(* CODESYS project cyber-gprs.20190329.3.project

Project tree, tasks and I/O mapping:
  Changsha_Xiangji_ARM_Cortex_A9_xilinx_zynq7000_linux : Changsha Xiangji-ARM Cortex A9(xilinx zynq7000)-linux, Changsha Xiangji Hiden Technology Co.Ltd, version 3.5.10.40
    application Application
      libraries: CAA Types Extern, 3.5.10.0 (CAA Technical Workgroup); VisuDialogs, * (System); CAA Real Time Clock Extern, 3.5.10.0 (CAA Technical Workgroup); CAA Callback Extern, 3.5.11.0 (CAA Technical Workgroup); CAA Can Low Level Extern, 3.5.11.0 (CAA Technical Workgroup); CAA Can Low Level Imp Extern, 3.5.11.0 (CAA Technical Workgroup); SysMem, 3.5.12.0 (System); CAA Net Base Services, 3.5.12.0 (CAA Technical Workgroup); CAA SerialCom, 3.5.12.0 (CAA Technical Workgroup); CAA File, 3.5.12.0 (CAA Technical Workgroup); CAA DTUtil Extern, 3.5.12.0 (CAA Technical Workgroup); SysFile, 3.5.9.0 (System); SysTypes2 Interfaces, * (System); Standard, * (System); cyber gpio, 3.5.10.40 (cyber); Util, * (System)
      task Task (cyclic, interval 50 ms, priority 0) calls prg_main
      task task_can (cyclic, interval 50 ms, priority 5) calls prg_can0, prg_can1, prg_test_can
      task EtherCAT_Task (cyclic, interval 10 ms, priority 1) calls nothing
      task VISU_TASK (cyclic, interval 100 ms, priority 31) calls VisuElems.Visu_Prg
      task Task_gprs (cyclic, interval 20 ms, priority 1) calls prg_heartbeat
      CAN_COMM/
        program prg_can0 [ST]: set_buf_18004f07, set_buf_18074f07, get_buf_0c00074f, proc_screen_data, set_buf_18104f07, set_buf_0801EE2A, get_buf_0C112AEE, set_buf_18114f07, set_buf_18044f07, set_buf_18024f07, set_buf_18014f07, get_buf_0c02074f, get_buf_0C132AEE, get_buf_0c05074f, get_buf_0c04074f, set_buf_18054f07, get_buf_0c01074f, get_buf_0C122AEE, set_buf_18124f07, set_buf_18084f07, set_buf_18064f07, set_buf_18144f07, set_buf_18094f07, set_buf_18034f07, set_buf_18134f07, get_buf_0c03074f, get_buf_0c07074f, get_buf_0c06074f
        program prg_can1 [ST]
        program prg_test_can [ST]
        function CAN_Send_MSG [ST]
      visualisation main
      program Test [ST]
      program Falsh_RW [ST]
      parameters/
        function fn_write_para_file [ST]
        function fn_read_para_file [ST]
        data type ST_PARA
      program prg_main [ST]
      global variables GVL
      funcs/
        function block FB_DOH_FAULT [ST]
        function is_hex [ST]
      program DO_fault [ST]
      GPRS/
        function block File_Read [ST]
        function Iccid_Get [ST]
        function block Packet_Heart [ST]
        program prg_heartbeat [ST]
        function block fb_get_iccid [ST]
        function block fb_m26 [ST]
        function block fb_get_lac [ST]
        function fn_cyber_layer1 [ST]
        function fn_cyber_layer2 [ST]
        function fn_cyber_heartBeat [ST]
        function fn_sn_str_to_byte [ST]
      gprs_lib/
        function block Com_Read [ST]
        function block reset_gprs [ST]
        function block Udp_Config [ST]
        function block Udp_Init [ST]
        function block UDP_Read [ST]
        function block Udp_Write [ST]
    IoDrvMIC7001 : IoDrvMIC7001, Cyber-MI, version 18.11.1
        input  Application.ai_20 : DWORD  // Ai20-Do02@C13
        input  Application.ai_21 : DWORD  // Ai21-Do03@C01
        input  Application.ai_22 : DWORD  // Ai22-Do04@C03
        input  Application.ai_23 : DWORD  // Ai23-Do05@C04
        input  Application.ai_24 : DWORD  // Ai24-Do06@C05
        input  Application.ai_25 : DWORD  // Ai25-Do07@C06
        input  Application.ai_26 : DWORD  // Ai26-Do08@C08
        input  Application.ai_27 : DWORD  // Ai27-Do09@C09
        input  Application.ai_28 : DWORD  // Ai28-Do10@C10
        input  Application.ai_29 : DWORD  // Ai29-Do11@C11
        input  Application.ai_30 : DWORD  // Ai30-Do12@D34
        input  Application.ai_31 : DWORD  // Ai31-Do13@D35
        input  Application.ai_34 : DWORD  // Ai34-Do16@D10
        input  Application.ai_35 : DWORD  // Ai35-Do17@D09
        input  Application.ai_36 : DWORD  // Ai36-Do18@D08
        input  Application.ai_37 : DWORD  // Ai37-Do19@D07
        input  Application.ai_38 : DWORD  // Ai38-Do20@D05
        input  Application.ai_39 : DWORD  // Ai39-Do21@D04
        input  Application.ai_40 : DWORD  // Ai40-Do22@D03
        input  Application.ai_41 : DWORD  // Ai41-Do23@D02
        input  Application.DI_cleanwater_LOW : DWORD  // Ai46-Ao00@C22
        input  Application.DI_Totvalve_Open : BOOL  // Di00-Ai00@C16
        input  Application.DI_water_overflow : BOOL  // Di02-Ai02@C17
        input  Application.DI_fog_pump_press_ok : BOOL  // Di05-Ai05@C19
        input  Application.DI_air_press_low : BOOL  // Di06-Ai06@C31
        input  Application.DI_Hpre_valve_open : BOOL  // Di07-Ai07@C20
        input  Application.DI_box_door_close : BOOL  // Di08-Ai08@C18
        input  Application.DI_backup_power_open : BOOL  // Di09-Ai09@D18
        input  Application.DI_Sweep_Down : BOOL  // Di10-Ai10@D20
        input  Application.DI_Rod_noDown : BOOL  // Di11-Ai11@D31
        input  Application.DI_Sweep_Up : BOOL  // Di12-Ai12@D19
        input  Application.DI_auxiliary2_warte_H : BOOL  // Di13-Ai13@D30
        input  Application.DI_auxiliary1_warte_H : BOOL  // Di14-Ai14@D29
        input  Application.DI_oil_release_valve : BOOL  // Di16-Ai16@D28
        input  Application.DI_Rcar : BOOL  // Di17-Ai17@D16
        input  Application.DI_oil_filter_block : BOOL  // Di18-Ai18@C25
        input  Application.DI_oil_level_low : BOOL  // Di19-Ai19@C24
        input  Application.DI_power_on : BOOL  // Di32-Ai32@D23
        input  Application.DI_sweep_out : BOOL  // Di33-Ai33@D12
        input  Application.DI_wastewater_full : BOOL  // Di42-Ai42@C23
        input  Application.DI_sweep_return : BOOL  // Di45-Ai45@D13
        output Application.DO_pointshoot_down : BOOL  // Do02-Ai20@C13
        output Application.DO_Lsweep_down : BOOL  // Do03-Ai21@C01
        output Application.DO_Lsweep_up : BOOL  // Do04-Ai22@C03
        output Application.DO_Rsweep_down : BOOL  // Do05-Ai23@C04
        output Application.DO_Rsweep_up : BOOL  // Do06-Ai24@C05
        output Application.DO_Lsweep_out : BOOL  // Do07-Ai25@C06
        output Application.DO_Rsweep_out : BOOL  // Do08-Ai26@C08
        output Application.DO_Lrod_out : BOOL  // Do09-Ai27@C09
        output Application.DO_Rrod_out : BOOL  // Do10-Ai28@C10
        output Application.DO_pointshoot_up : BOOL  // Do11-Ai29@C11
        output Application.DO_backup_power : BOOL  // Do12-Ai30@D34
        output Application.DO_Motor_en : BOOL  // Do13-Ai31@D35
        output Application.DO_fog_Spump : BOOL  // Do16-Ai34@D10
        output Application.DO_Hpre_pump : BOOL  // Do17-Ai35@D09
        output Application.DO_selfclean_water : BOOL  // Do18-Ai36@D08
        output Application.DO_Hpressure_water : BOOL  // Do19-Ai37@D07
        output Application.DO_Suction_water : BOOL  // Do20-Ai38@D05
        output Application.DO_Rrod_water : BOOL  // Do21-Ai39@D04
        output Application.DO_Lrod_water : BOOL  // Do22-Ai40@D03
        output Application.DO_water_overflow : BOOL  // Do23-Ai41@D02
        output Application.DO_pointshoot_left : BOOL  // Do28-Pwmi00@C33
        output Application.DO_pointshoot_right : BOOL  // Do29-Pwmi01@C34
        output Application.DO_watercooler_pump : BOOL  // Do30-Pwmi02@D25
        output Application.DO_cooler_fan : BOOL  // Do31-Pwmi03@D26
        unmapped channels: Ai00@C16, Ai01@C28, Ai02@C17, Ai03@C29, Ai04@C30, Ai05@C19, Ai06@C31, Ai07@C20, Ai08@C18, Ai09@D18, Ai10@D20, Ai11@D31, Ai12@D19, Ai13@D30, Ai14@D29, Ai15@D17, Ai16@D28, Ai17@D16, Ai18-Do00@C25, Ai19-Do01@C24, Ai32-Do14@D23, Ai33-Do15@D12, Ai42-Do24@C23, Ai43-Do25@C35, Ai44-Do26@D24, Ai45-Do27@D13, Ai47-Ao01@D14, Ai48_Pi02, Ai49_Out5V, Ai50_VCC, Ai51_VCC_L, Ai52_VCC_R, Ai53_Pwm-i0, Ai54_Pwm-i1, Ai55_Pwm-i2, Ai56_Pwm-i3, Ai57_CPU-T, Ai58_G-x, Ai59_G-y, Ai60_G-z,
          Ai61-reserved, Ai62-IO-cntr, Ai63-CDS-cntr, Di01-Ai01@C28, Di03-Ai03@C29, Di04-Ai04@C30, Di15-Ai15@D17, Di20-Ai20@C13, Di21-Ai21@C01, Di22-Ai22@C03, Di23-Ai23@C04, Di24-Ai24@C05, Di25-Ai25@C06, Di26-Ai26@C08, Di27-Ai27@C09, Di28-Ai28@C10, Di29-Ai29@C11, Di30-Ai30@D34, Di31-Ai31@D35, Di34-Ai34@D10, Di35-Ai35@D09, Di36-Ai36@D08, Di37-Ai37@D07, Di38-Ai38@D05, Di39-Ai39@D04, Di40-Ai40@D03, Di41-Ai41@D02, Di43-Ai43@C35, Di44-Ai44@D24, Di46-Ai46@C22, Di47-Ai47@D14, Di48-Pi00@C15, Di49-Pi01@C14, Di50-Pi02@D22, Di51-Pi03@D21, Di52-reserved, Di53-reserved, Di54-reserved, Di55-reserved, Di56-reserved,
          Di57-reserved, Di58-reserved, Di59-reserved, Di60-reserved, Di61-reserved, Di62-reserved, Di63-reserved, Pi00-Di48@C15, Pi01-Di49@C14, Pi02-Di50@D22, Pi03-Di51@D21, Do00-Ai18@C25, Do01-Ai19@C24, Do14-Ai32@D23, Do15-Ai33@D12, Do24-Ai42@C23, Do25-Ai43@C35, Do26-Ai44@D24, Do27-Ai45@D13, PWM00@C25, PWM01@C24, PWM02@C13, PWM03@C01, PWM04@C03, PWM05@C04, PWM06@C05, PWM07@C06, PWM08@C08, PWM09@C09, PWM10@C10, PWM11@C11, PWM12@D34, PWM13@D35, PWM14@D23, PWM15@D12, PWM16@D10, PWM17@D09, PWM18@D08, PWM19@D07, PWM20@D05,
          PWM21@D04, PWM22@D03, PWM23@D02, PWM24@C23, PWM25@C35, PWM26@D24, PWM27@D13, PWM28-Pwmi00@C33, PWM29-Pwmi01@C34, PWM30-Pwmi02@D25, PWM31-Pwmi03@D26, PWM_I_0@C33, PWM_I_1@C34, PWM_I_2@D25, PWM_I_3@D26, Ao00-Ai46@C22, Ao01-Ai47@D14, LED_run, LED_err, LED_usr, ctrl_ai_raw, ctrl_adjust, ctrl_adj0, ctrl_adj1, ctrl_adj2, ctrl_adj3, ctrl_adj4
    SoftMotion General Axis Pool
    EtherCAT_Master_SoftMotion : EtherCAT Master SoftMotion, 3S - Smart Software Solutions GmbH, version 3.5.12.40
        settings: MasterCycleTime = 10000; SlaveAutoRestart = True; NetworkName = 'eth0'; NetworkName = "eth0"; SelectNetworkByName = True; SrcAddress1 = 29185; SrcAddress2 = 102470395
      MIR3501 : MIR3501, xiangrui, order no. MIR3501, version Revision=16#00000000
          settings: StationAlias = 0; DC sync0 cycletime = 10000; DC sync1 cycletime = 10000
          output Application.DO_wastewater_valve : BIT  // DO-00-C01
          output Application.DO_wastewater_pump : BIT  // DO-01-C02
          output Application.DO_oil_release_valve : BIT  // DO-02-C03
          output Application.DO_Sweep_Mspeed : BIT  // DO-03-C04
          output Application.DO_Sweep_Lspeed : BIT  // DO-04-C05
          output Application.DO_RSweep : BIT  // DO-05-C06
          output Application.DO_LASweep : BIT  // DO-06-C07
          output Application.DO_RASweep : BIT  // DO-07-C08
          output Application.DO_Box_Down : BIT  // DO-08-C09
          output Application.DO_Suction_Down : BIT  // DO-10-C11
          output Application.DO_Suction_Up : BIT  // DO-11-C12
          output Application.DO_Door_Close : BIT  // DO-12-C26
          output Application.DO_Door_Open : BIT  // DO-13-C25
          output Application.DO_Box_Up : BIT  // DO-15-C33
          unmapped channels: DO-09-C10, DO-14-C34, PWM-00-C26, PWM-01-C25, PWM-02-C34, PWM-03-C33, PWMi-00-C26, PWMi-01-C25, PWMi-02-C34, PWMi-03-C33, AI-00-C17, AI-01-C29, AI-02-C18, AI-03-C30, AI-04-C14, AI-05-C15, AI-06-C21, AI-07-C22, AI-08-C01, AI-09-C02, AI-10-C03, AI-11-C04, AI-12-C05, AI-13-C06, AI-14-C07, AI-15-C08, AI-16-C09, AI-17-C10, AI-18-C11, AI-19-C12, AI-20, AI-21, AI-22, AI-23, DI-00-C17, DI-01-C29, DI-02-C18, DI-03-C30, DI-04-C14, DI-05-C15,
            DI-06-C21, DI-07-C22, DI-08-C01, DI-09-C02, DI-10-C03, DI-11-C04, DI-12-C05, DI-13-C06, DI-14-C07, DI-15-C08, DI-16-C09, DI-17-C10, DI-18-C11, DI-19-C12, DI-20-C27, DI-21-C16, DI-22-C19, DI-23-C20, DI-24, DI-25, DI-26, DI-27, DI-28, DI-29, DI-30, DI-31, PI-00-C27, PI-01-C16, PI-02-C19, PI-03-C20
  5ce3da45-db07-42e7-a21c-a00fff4ed8f6|C:\Users\Administrator\Desktop\robotview1.bmp
  5ce3da45-db07-42e7-a21c-a00fff4ed8f6|C:\Users\Administrator\Desktop\robotview2.bmp
  text list GlobalTextList
  5ce3da45-db07-42e7-a21c-a00fff4ed8f6|C:\Users\Administrator\Desktop\1129.bmp
  5ce3da45-db07-42e7-a21c-a00fff4ed8f6|C:\Users\Administrator\Desktop\robotview0.bmp
*)

// Changsha_Xiangji_ARM_Cortex_A9_xilinx_zynq7000_linux/Application/parameters/ST_PARA
TYPE ST_PARA :
STRUCT
	len:UINT := 64;   //参数的个数，根据需要设置。设置后最好不变，改变后以前保存的参数作废
	para_val:ARRAY[0..63] OF REAL; 	
	para_ok:BOOL := FALSE;
END_STRUCT
END_TYPE

// Changsha_Xiangji_ARM_Cortex_A9_xilinx_zynq7000_linux/Application/GVL
VAR_GLOBAL
	g_parameters: ST_PARA;	
	
	//通过CAN总线从底盘读到的信息
	High_voltage_Ready:BOOL := FALSE;
	Chassis_speed:BYTE := 0;
	Chassis_Soc:BYTE := 0;
//********以下为显示屏下发指令*********//
    // 全洗扫
	HMI_Awashsweep: BOOL := FALSE;	
    // 左洗扫
	HMI_Lwashsweep: BOOL := FALSE;	
    // 右洗扫
	HMI_Rwashsweep: BOOL := FALSE;
	// 全扫路
	HMI_Asweeproad: BOOL := FALSE;
	// 左扫路
	HMI_Lsweeproad: BOOL := FALSE;
	// 右扫路
	HMI_Rsweeproad: BOOL := FALSE;
	// 全清洗
	HMI_Acleanwash: BOOL := FALSE;
	// 右清洗
	HMI_Lcleanwash: BOOL := FALSE;
	// 右全洗
	HMI_Rcleanwash: BOOL := FALSE;
	// 停扫
	HMI_stop_sweep: BOOL := FALSE;
	// 电机启动
	HMI_start_motor: BOOL := FALSE;
	// 电机停止
	HMI_stop_motor: BOOL := FALSE;
	// 速度加
	HMI_Inc_Speed: BOOL := FALSE;
	// 速度减
	HMI_Dec_Speed: BOOL := FALSE;
	// 标准转速
	HMI_Standard_speed: BOOL := FALSE;
	// 强力转速
	HMI_Strong_speed: BOOL := FALSE;
	// 箱门关
	HMI_Door_Close: BOOL := FALSE;
	// 箱门开
	HMI_Door_Open: BOOL := FALSE;
	// 箱体升
	HMI_Box_Up: BOOL := FALSE;
	// 箱体降
	HMI_Box_Down: BOOL := FALSE;
	// 喷雾降尘泵
	HMI_fog_Spump: BOOL := FALSE;
	// 自洁
	HMI_selfclean: BOOL := FALSE;
	// 污水泵
	HMI_wastewater_pump: BOOL := FALSE;
	// 扫盘高速
	HMI_Sweep_Hspd: BOOL := FALSE;
	// 扫盘中速
	HMI_Sweep_Mspd: BOOL := FALSE;
	// 扫盘低速
	HMI_Sweep_Lspd: BOOL := FALSE;
	// 高压冲洗
	HMI_Hpre_wash: BOOL := FALSE;
	// 点喷上
	HMI_pointshoot_up: BOOL := FALSE;
	// 点喷下
	HMI_pointshoot_down: BOOL := FALSE;
	// 点喷左
	HMI_pointshoot_left: BOOL := FALSE;
	// 点喷右
	HMI_pointshoot_right: BOOL := FALSE;
	// 排水启动
	HMI_drain_start: BOOL := FALSE;
	// 排水自动
	HMI_drain_auto: BOOL := FALSE;
	// 排水手动
	HMI_drain_manual: BOOL := FALSE;
	// 左喷杆排水
	HMI_Lrod_drain: BOOL := FALSE;
	// 右喷杆排水
	HMI_Rrod_drain: BOOL := FALSE;
	// 高辅排水
	HMI_Hpressure_drain: BOOL := FALSE;
	// 自洁排水
	HMI_selfclean_drain: BOOL := FALSE;
	// 吸嘴排水
	HMI_Suction_drain: BOOL := FALSE;
	// 功能测试
	HMI_func_test: BOOL := FALSE;
	// 更换扫刷
	HMI_replace_Sweep: BOOL := FALSE;
	// 智能
	HMI_intelligent: BOOL := FALSE;
	// 清洁
	HMI_cleanly: BOOL := FALSE;
	// 一般
	HMI_normal: BOOL := FALSE;
	// 污染
	HMI_dirty: BOOL := FALSE;
	// 水冷泵测试
	Test_watercooler_pump: BOOL := FALSE;
	// 散热风扇测试
	Test_cooler_fan: BOOL := FALSE;
	// 扫盘中速
	Test_Sweep_Mspeed: BOOL := FALSE;
	// 扫盘低速
	Test_Sweep_Lspeed: BOOL := FALSE;
	// 左扫旋转
	Test_LSweep: BOOL := FALSE;
	// 右扫旋转
	Test_RSweep: BOOL := FALSE;
	// 全扫旋转
	Test_ASweep: BOOL := FALSE;
	// 箱体降
	Test_Box_Down: BOOL := FALSE;
	// 箱体升
	Test_Box_Up: BOOL := FALSE;
	// 吸嘴下降
	Test_Suction_Down: BOOL := FALSE;
	// 吸嘴上升
	Test_Suction_Up: BOOL := FALSE;
	// 箱门开
	Test_Door_Open: BOOL := FALSE;
	// 箱门关
	Test_Door_Close: BOOL := FALSE;
	// 左扫盘下降
	Test_LSweep_Down: BOOL := FALSE;
	// 左扫盘上升
	Test_LSweep_Up: BOOL := FALSE;
	// 右扫盘下降
	Test_RSweep_Down: BOOL := FALSE;
	// 右扫盘上升
	Test_RSweep_Up: BOOL := FALSE;
	// 左扫盘摆出
	Test_LSweep_out: BOOL := FALSE;
	// 右扫盘摆出
	Test_RSweep_out: BOOL := FALSE;
	// 左喷杆摆出
	Test_Lrod_OUT: BOOL := FALSE;
	// 右喷杆摆出
	Test_Rrod_OUT: BOOL := FALSE;
	// 左喷杆喷水
	Test_Lrod_water: BOOL := FALSE;
	// 右喷杆喷水
	Test_Rrod_water: BOOL := FALSE;
	// 吸嘴喷杆喷水
	Test_Suction_water: BOOL := FALSE;
	// 高压喷杆喷水
	Test_Hpre_wash: BOOL := FALSE;
	// 自洁
	Test_selfclean: BOOL := FALSE;
	// 高压水泵啮合
	Test_Hpre_pump_gearin: BOOL := FALSE;
	// 喷雾降尘泵
	Test_fogpump: BOOL := FALSE;
	// 点喷上
	Test_pointshoot_up: BOOL := FALSE;
	// 点喷下
	Test_pointshoot_down: BOOL := FALSE;
	// 点喷左
	Test_pointshoot_left: BOOL := FALSE;
	// 点喷右
	Test_pointshoot_right: BOOL := FALSE;
	// 污水泵
	Test_wastewater_pump: BOOL := FALSE;
	// 污水球阀
	Test_wastewater_valve: BOOL := FALSE;
	// 备用动力打开
	Test_backup_power: BOOL := FALSE;
	// 转速加减值
	Re_IncDec_Speed: UINT;
	// 电机最低转速
	Re_motor_min_speed: UINT;
	// 标准转速
	Re_normal_speed: UINT;
	// 强力转速
	Re_strong_Speed: UINT;
	// 扫盘转速
	Re_Sweep_Speed: UINT;
	// 高压水泵超速报警
	Re_Pumpspeed_arm: UINT;
	// 高压水泵超速停止
	Re_Pumpspeed_stop: UINT;
	// 电机最高转速
	Re_MAX_Speed: UINT;
	// 电机怠速
	Re_Idle_Speed: UINT;	
    // 清洁低速
	Re_clean_low_speed: UINT;
	// 清洁中低速
	Re_clean_midlow_speed: UINT;
	// 清洁中高速
	Re_clean_midhigh_speed: UINT;
	// 清洁高速
	Re_clean_high_speed: UINT;
	// 一般低速
	Re_normal_low_speed: UINT;
	// 一般中低速
	Re_normal_midlow_speed: UINT;
	// 一般中高速
	Re_normal_midhigh_speed: UINT;
	// 一般高速
	Re_normal_high_speed: UINT;
	// 污染低速
	Re_dirty_low_speed: UINT;
	// 污染中低速
	Re_dirty_midlow_speed: UINT;
	// 污染中高速
	Re_dirty_midhigh_speed: UINT;
	// 污染高速
	Re_dirty_high_speed: UINT;
	//************************************
	//********以下为控制器输出**********//
	//***********************************
	// 左扫盘下降
	DO_Lsweep_down: BOOL;
	// 左扫盘上升
	DO_Lsweep_up: BOOL;
	// 右扫盘下降
	DO_Rsweep_down: BOOL;
	// 右扫盘上升
	DO_Rsweep_up: BOOL;
	// 左扫盘摆出
	DO_Lsweep_out: BOOL;
	// 右扫盘摆出
	DO_Rsweep_out: BOOL;
	// 左喷杆摆出
	DO_Lrod_out: BOOL;
	// 右喷杆摆出
	DO_Rrod_out: BOOL;
	// 点喷上
	DO_pointshoot_up: BOOL;
	// 点喷下
	DO_pointshoot_down: BOOL;
	// 点喷左
	DO_pointshoot_left: BOOL;
	// 点喷右
	DO_pointshoot_right: BOOL;
	// 水路卸荷阀
	DO_water_overflow: BOOL;
	// 左喷杆喷水
	DO_Lrod_water: BOOL;
	// 右喷杆喷水
	DO_Rrod_water: BOOL;
	// 吸嘴喷杆喷水
	DO_Suction_water: BOOL;
	// 喷雾喷杆喷水
	DO_Hpressure_water: BOOL;
	// 自洁喷水
	DO_selfclean_water: BOOL;
	// 低压隔膜泵
	DO_fog_Spump: BOOL;
	// 高压水泵啮合
	DO_Hpre_pump: BOOL;
	// 电机使能
	DO_Motor_en: BOOL;
	// 水冷泵打开
	DO_watercooler_pump: BOOL;
	// 散热风扇打开
	DO_cooler_fan: BOOL;
	// 备用动力打开
	DO_backup_power: BOOL;
	// 污水泵球阀打开
	DO_wastewater_valve: BOOL;
	// 污水泵打开
	DO_wastewater_pump: BOOL;
	// 油路卸荷阀
	DO_oil_release_valve: BOOL;
	// 扫盘中速
	DO_Sweep_Mspeed: BOOL;
	// 扫盘低速
	DO_Sweep_Lspeed: BOOL;
	// 右扫旋转
	DO_RSweep: BOOL;
	// 左/全扫旋转
	DO_LASweep: BOOL;
	// 右/全扫旋转
	DO_RASweep: BOOL;
	// 箱体降
	DO_Box_Down: BOOL;
	// 箱体升
	DO_Box_Up: BOOL;
	// 吸盘下降
	DO_Suction_Down: BOOL;
	// 吸盘上升
	DO_Suction_Up: BOOL;
	// 箱门打开
	DO_Door_Open: BOOL;
	// 箱门关闭
	DO_Door_Close: BOOL;
	// 高压水泵啮合
	DO_Hpre_pump1: BOOL;
	// 左扫盘摆出中间变量
	DO_Lsweep_out1: BOOL;
	// 左扫盘下降中间变量
	DO_Lsweep_down1: BOOL;
	// 右扫盘摆出中间变量
	DO_Rsweep_out1: BOOL;
	// 右扫盘下降中间变量
	DO_Rsweep_down1: BOOL;
	// 吸盘下降中间变量
	DO_Suction_Down1: BOOL;
	// 右扫盘上升标志
	DO_Rsweep_up1: BOOL;
	// 吸盘上升标志位
	DO_Suction_Up1: BOOL;
	// 左喷杆摆出标志
	DO_Lrod_out1: BOOL;
	// 右喷杆摆出标志位
	DO_Rrod_out1: BOOL;
	// 喷雾降尘泵标志位
	DO_fog_Spump1: BOOL;
	// 高压冲洗标志位
	DO_Hpressure_water1: BOOL;
	// 自洁标志位
	DO_selfclean_water1: BOOL;
	// 垃圾箱门关标志位
	DO_Door_Close1: BOOL;
	// 垃圾箱门开标志位
	DO_Door_Open1: BOOL;
	// 箱体升标志
	DO_Box_Up1: BOOL;
	// 垃圾箱下降标志
	DO_Box_Down1: BOOL;
	// 水冷泵电机打开标志位
	DO_watercooler_pump_open1: BOOL;
	// 散热风扇打开标志位
	DO_cooler_fan_open1: BOOL;
	
	//********控制器输入**************
	//**********************************
	// 水箱水位低
	DI_cleanwater_LOW: DWORD;
	// 总水阀打开
	DI_Totvalve_Open: BOOL;
	// 箱门关闭
	DI_box_door_close: BOOL;
	// 高压吹净球阀打开
	DI_Hpre_valve_open: BOOL;

	// 污水满
	DI_wastewater_full: BOOL;
	// 撑杆未放下
	DI_Rod_noDown: BOOL;
	// 备用动力开
	DI_backup_power_open: BOOL;
	// 水路卸荷阀卸荷
	DI_water_overflow: BOOL;

	// 电源开关打开
	DI_power_on: BOOL;
	// 倒车
	DI_Rcar: BOOL;
	// 液压卸荷阀
	DI_oil_release_valve: BOOL;
	// 辅污水箱1水位高
	DI_auxiliary1_warte_H: BOOL;
	// 辅污水箱2水位高
	DI_auxiliary2_warte_H: BOOL;
	// 扫盘升
	DI_Sweep_Up: BOOL;
	// 扫盘降
	DI_Sweep_Down: BOOL;
	// 扫盘摆出
	DI_sweep_out: BOOL;
	// 扫盘缩回
	DI_sweep_return: BOOL;
	// 全洗扫标志位
	AwashSweep_HMI: BOOL := FALSE;
	// 左洗扫标志位
	LwashSweep_HMI: BOOL := FALSE;
	// 右洗扫标志位
	RwashSweep_HMI: BOOL := FALSE;
	// 全扫路标志位
	ASweeproad_HMI: BOOL := FALSE;
	// 左扫路标志位
	LSweeproad_HMI: BOOL := FALSE;
	// 右扫路标志位
	RSweeproad_HMI: BOOL := FALSE;
	// 全清洗标志位
	Aclean_HMI: BOOL := FALSE;
	// 左清洗标志位
	Lclean_HMI: BOOL := FALSE;
	// 右清洗标志位
	Rclean_HMI: BOOL := FALSE;
	// 停扫标志位
	Sweep_stop_HMI: BOOL := FALSE;
	// 标准转速标志位
	Standard_speed_HMI: BOOL := FALSE;
	// 强力转速
	Strong_speed_HMI: BOOL := FALSE;
	// 扫盘高速
	Sweep_HSpeed_HMI: BOOL;
	// 扫盘中速
	Sweep_MSpeed_HMI: BOOL;
	// 扫盘低速
	Sweep_LSpeed_HMI: BOOL;
	// 排水启动
	Drain_start_HMI: BOOL := FALSE;
	// 排水自动
	Drain_auto_HMI: BOOL;
	// 排水手动
	Drain_manual_HMI: BOOL;
	// 左喷杆排水
	Lrod_drain_HMI: BOOL;
	// 右喷杆排水
	Rrod_drain_HMI: BOOL;
	// 高辅排水
	Hpressure_drain_HMI: BOOL;
	// 自洁排水
	Selfclean_drain_HMI: BOOL;
	// 吸嘴喷杆排水
	Suction_drain_HMI: BOOL;
	// 更换扫刷标志位
	replace_Sweep_HMI: BOOL;
	// 功能测试
	Func_test_HMI: BOOL;
	// 智能标志位
	Intelligent_HMI: BOOL:= FALSE;
	// 清洁标志位
	Cleanly_HMI: BOOL:= FALSE;
	// 一般标志位
	Normal_HMI: BOOL:= FALSE;
	// 污染标志位
	Dirty_HMI: BOOL:= FALSE;

	// 点喷上标志位
	Pointshoot_up_HMI: BOOL;
	// 点喷下标志位
	Pointshoot_down_HMI: BOOL;
	// 点喷左标志位
	Pointshoot_left_HMI: BOOL;
	// 点喷右标志位
	Pointshoot_right_HMI: BOOL;
	// 水冷泵测试标志位
	cooler_motor_Test: BOOL;
	// 散热风扇测试标志位
	cooler_fan_Test: BOOL;
	// 扫盘中速测试标志位
	Sweep_Mspeed_Test: BOOL;
	// 扫盘低速测试标志位
	Sweep_Lspeed_Test: BOOL;
	// 左扫旋转测试标志位
	LSweep_Test: BOOL;
	// 右扫测试标志位
	RSweep_Test: BOOL;
	// 全扫测试标志位
	ASweep_Test: BOOL;
	// 箱体降测试标志位
	Box_Down_Test: BOOL;
	// 箱体升测试标志位
	Box_Up_Test: BOOL;
	// 吸盘降测试标志位
	Suction_Down_Test: BOOL;
	// 吸盘升测试标志位
	Suction_Up_Test: BOOL;
	// 箱门开测试标志位
	Boxdoor_open_Test: BOOL;
	// 测试标志位
	Boxdoor_close_Test: BOOL;
	// 左扫降测试标志位
	LSweep_Down_Test: BOOL;
	// 左扫升测试标志位
	LSweep_Up_Test: BOOL;
	// 右扫降测试标志位
	RSweep_Down_Test: BOOL;
	// 右扫升测试标志位
	RSweep_Up_Test: BOOL;
	// 左扫摆出测试标志位
	Lrod_OUT_Test: BOOL;
	// 右扫摆出测试标志位
	Rrod_OUT_Test: BOOL;
	// 左喷杆喷水测试标志位
	Lrod_water_Test: BOOL;
	// 右喷杆喷水测试标志位
	Rrod_water_Test: BOOL;
	// 吸嘴喷水测试标志位
	Suction_water_Test: BOOL;
	// 高辅喷水测试标志位
	Hpre_wash_Test: BOOL;
	// 自洁测试标志位
	selfclean_water_Test: BOOL;
	// 高压水泵啮合测试标志位
	Hpress_pump_gearin_Test: BOOL;
	// 喷雾降尘测试标志位
	Fog_pump_Test: BOOL;
	// 左扫摆出测试标志位
	LSweep_out_Test: BOOL;
	// 右扫摆出测试标志位
	RSweep_out_Test: BOOL;
	// 污水泵测试标志位
	Wastewater_pump_Test: BOOL;
	// 污水泵球阀测试标志位
	Wastewater_valve_Test: BOOL;
	// 备用动力测试标志位
	Backup_power_Test: BOOL;
	// 点喷上测试标志位
	Pointshoot_up_Test: BOOL;
	// 点喷下测试标志位
	Pointshoot_down_Test: BOOL;
	// 点喷左测试标志位
	Pointshoot_left_Test: BOOL;
	// 点喷右测试标志位
	Pointshoot_right_Test: BOOL;
	// 电机工作标志位
	Motor_Work: BOOL:= FALSE;
	// 系统工作标志位
	SYS_work: BOOL;
	// 转速加减值
	S_IncDec_Speed: UINT;
	// 电机最低转速
	S_min_speed: UINT;
	// 标准转速
	S_Standard_Speed: UINT;
	// 强力转速
	S_Strong_Speed: UINT;
	// 扫盘转速
	S_Sweep_Speed: UINT;
	// 高压水泵超速报警
	S_Pumpspeed_arm: UINT;
	// 高压水泵超速停止
	S_Pumpspeed_stop: UINT;
	// 最高转速
	S_MAX_Speed: UINT;
	// 电机怠速
	S_Idle_Speed: UINT;
	// 电机实际转矩
	Motor_real_torque_HMI: UINT;
	// 电机实际转速
	Motor_real_speed_HMI: UINT;
	// 电机母线电压
	Motor_bus_voltage_HMI: UINT;
	// 电机相电流
	Motor_phase_current_HMI: UINT;
	// 电机最大允许驱动转矩
	Motor_max_dirve_torque_HMI: UINT;
	// 电机最大允许制动转矩
	Motor_max_brake_torque_HMI: UINT;
	// 电机驱动器温度
	Motor_temp_controller_HMI: BYTE;
	// 电机温度
	Motor_temp_HMI: BYTE;
	// 电机最大转速
	Motor_max_speed_HMI: UINT;
	// 电机运行方向
	Motor_direction_cw: BYTE;
	// 电机工作模式
	Motor_mode: BYTE;
	// 电机状态
	Motor_stat: BYTE;
	// 电机母线欠压
	Motor_bus_low_voltage: BYTE;
	// 电机母线欠压
	Motor_bus_high_voltage: BYTE;
	// 电机控制器过温
	MOtor_ctrller_high_temp: BYTE;
	// 电机过温
	Motor_high_temp: BYTE;
	// 电机IGBT故障
	Motor_igbt_fault: BYTE;
	// 电机超速
	Motor_overspeed: BYTE;
	// 电机通讯故障
	Motor_comm_error: BYTE;
	// 电机过流或短路
	Motor_short: BYTE;
	// 电机堵转故障
	Motor_overload: BYTE;
	// 电机自检故障
	Motor_selfcheck_fault: BYTE;
	// 电机低压供电故障
	Motor_low_voltage: BYTE;
	// 电机传感器故障
	Motor_sensor_fault: BYTE;

	// 设定转速值
	SETspeed_PID: UINT:= 0;
	// 底盘车速
//	Chassis_speed: UINT;
	// 清洁路面低速
	S_clean_low_speed: UINT;
	// 清洁中低速
	S_clean_midlow_speed: UINT;
	// 清洁中高速
	S_clean_midhigh_speed: UINT;
	// 清洁高速
	S_clean_high_speed: UINT;
	// 一般路面低速
	S_normal_low_speed: UINT;
	// 一般路面中低速
	S_normal_midlow_speed: UINT;
	// 一般路面中高速
	S_normal_midhigh_speed: UINT;
	// 一般路面高速
	S_normal_high_speed: UINT;
	// 污染路面低速
	S_dirty_low_speed: UINT;
	// 污染路面中低速
	S_dirty_midlow_speed: UINT;
	// 污染路面中高速
	S_dirty_midhigh_speed: UINT;
	// 污染路面高速
	S_dirty_high_speed: UINT;
	// 水箱水位低报警
	DI_cleanwater_LOW_ALM: BOOL;
	// 请先打开备用动力开关
	Backup_power_Test_warn: BOOL;
	// 水路卸荷阀未关闭故障
	T_water_overflow_noClose: Ton;
	// 水路卸荷阀未打开故障
	T_water_overflow_noOpen: Ton;
	// 喷雾降尘泵压力不正常标志
	T_fog_pump_press_noOk: Ton;
	// 主污水箱水满标志
	T_DI_wastewater_full: Ton;
	// 辅污水箱1水满标志
	T_DI_auxiliary1_warte_H: Ton;
	// 辅污水箱2水满标志
	T_DI_auxiliary2_warte_H: Ton;
	// 污水满故障标志
	Wastewater_full_Fault: BOOL;
	// 辅助水箱水位不一致标志
	T_auxiliary_warte_dif: Ton;
	// 回油过滤堵塞故障标志
	T_DI_oil_filter_block: Ton;
	// 液压油位低故障标志
	T_DI_oil_level_low: Ton;
	// 系统气压低标志
	T_DI_air_press_low: Ton;
	// 倒车标志
	T_DI_Rcar: Ton;
	// 水箱缺水故障标志
	T_DI_cleanwater_LOW: Ton;
	// 高压水泵超速报警
	T_Pumpspeed_H: Ton;
	// 高压水泵超速停止
	T_Pumpspeed_HH: Ton;
	// 请关闭测试提示
	TEST_ALM: BOOL;
	// 倒车提示
	RCAR_ALM: BOOL;
	// 请先打开发动机
	Motor_Work_ALM: BOOL;
	// 倒车故障停机
	DI_Rcar_fault: BOOL;
	// 污水满故障停机
	Wastewater_full_Fault1: BOOL;
	// 底盘电量低于20%
	Chassis_SOC_LOW: BOOL;
	// 底盘电量低7S后停机
	T_Chassis_SOC_LOW: Ton;
	// 隔膜泵球阀未打开
	fog_Spump_arm: BOOL;
	// 污水泵打开标志位
	DO_wastewater_pump_open1: BOOL;
	// 高压水泵未啮合提示
	DO_Hpre_pump_noWork: BOOL;
	// 高压水路球阀未打开提示
	DI_Totvalve_noOpen: BOOL;
	// 高压吹净球阀未打开提示
	DI_Hpre_valve_noOpen: BOOL;
	// 请先打开箱门
	DO_Box_Up_arm: BOOL;
	// 请先放下撑杆
	DO_Box_Down_arm: BOOL;
	// 底盘未上高压提示
	High_voltage_noReady: BOOL;
	// 故障停机
	Fault_STOP: BOOL;
	// 底盘CAN通信故障
	T_Chassis_CAN_fault: TON;
	// 与电机CAN通讯失败
	T_Motor_CAN_fault: Ton;
	// 与屏CAN通讯失败
	T_Screen_CAN_fault: Ton;
	// 屏通讯失败停扫
	HMI_MOTOR_runstop_M: BOOL;
	// 全扫旋转标志
	ASweep: BOOL;
	// 左扫旋转标志
	LSweep: BOOL;
	// 右扫旋转标志
	RSweep: BOOL;
	

	// 喷雾降尘泵压力正常
	DI_fog_pump_press_ok: BOOL;
	// 液压油位低
	DI_oil_level_low: BOOL;
	// 回油过滤堵塞
	DI_oil_filter_block: BOOL;
	// 气路系统压力低
	DI_air_press_low: BOOL;
	Drain_manual_HMI100: BOOL;
	ai_21: DWORD;
	ai_22: DWORD;
	ai_23: DWORD;
	ai_24: DWORD;
	ai_25: DWORD;
	ai_26: DWORD;
	ai_27: DWORD;
	ai_28: DWORD;
	ai_29: DWORD;
	ai_20: DWORD;
	ai_41: DWORD;
	ai_40: DWORD;
	ai_39: DWORD;
	ai_38: DWORD;
	ai_37: DWORD;
	ai_36: DWORD;
	ai_35: DWORD;
	ai_34: DWORD;
	ai_31: DWORD;
	ai_30: DWORD;
					
	DO_Lsweep_down_short: BOOL:= FALSE;  //左扫盘降短路标志
	DO_Lsweep_down_open: BOOL := FALSE;   //左扫盘降开路标志
	DO_Lsweep_up_short: BOOL := FALSE;  // 左扫盘升短路标志
	DO_Lsweep_up_open: BOOL := FALSE;   //左扫盘升开路标志
	DO_Rsweep_down_short: BOOL:= FALSE; //右扫盘降短路
	DO_Rsweep_down_open: BOOL:= FALSE; //右扫盘降开路
	DO_Rsweep_up_short: BOOL:= FALSE; //右扫盘升短路
	DO_Rsweep_up_open: BOOL:= FALSE; //右扫盘升开路
	DO_Lsweep_out_short: BOOL:= FALSE; //左扫摆出短路
	DO_Lsweep_out_open: BOOL:= FALSE; //左扫摆出开路
	DO_Rsweep_out_short: BOOL:= FALSE; //右扫盘摆出短路
	DO_Rsweep_out_open: BOOL:= FALSE; //右扫盘摆出开路
	DO_Lrod_out_short: BOOL:= FALSE; //左喷杆摆出短路
	DO_Lrod_out_open: BOOL:= FALSE; //左喷杆摆出开路
	DO_Rrod_out_short: BOOL:= FALSE; //右喷杆摆出短路
	DO_Rrod_out_open: BOOL:= FALSE; //右喷杆摆出开路
	DO_pointshoot_up_short: BOOL:= FALSE; //点喷上短路
	DO_pointshoot_up_open: BOOL:= FALSE; //点喷上开路
	DO_pointshoot_Down_short: BOOL:= FALSE; //点喷下短路
	DO_pointshoot_Down_open: BOOL:= FALSE; //点喷下开路
	DO_pointshoot_left_short: BOOL:= FALSE; //点喷左短路
	DO_pointshoot_left_open: BOOL:= FALSE; //点喷左开路
	DO_pointshoot_right_short: BOOL:= FALSE; //点喷右短路
	DO_pointshoot_right_open: BOOL:= FALSE; //点喷右开路
	DO_water_overflow_short: BOOL:= FALSE; //水路卸荷阀短路
	DO_water_overflow_open: BOOL:= FALSE; //水路卸荷阀开路
	DO_Lrod_water_short: BOOL:= FALSE; //左侧喷杆球阀打开短路
	DO_Lrod_water_open: BOOL:= FALSE; //左侧喷杆球阀打开开路
	DO_Rrod_water_short: BOOL:= FALSE; //右侧喷杆球阀打开短路
	DO_Rrod_water_open: BOOL:= FALSE; //右侧喷杆球阀打开开路
	DO_Suction_water_short: BOOL:= FALSE; //吸嘴喷杆球阀打开短路
	DO_Suction_water_open: BOOL:= FALSE; //吸嘴喷杆球阀打开开路
	DO_Hpressure_water_short: BOOL:= FALSE; //喷雾球阀打开短路
	DO_Hpressure_water_open: BOOL:= FALSE; //喷雾球阀打开开路
	DO_selfclean_water_short: BOOL:= FALSE; //自洁喷杆球阀打开短路
	DO_selfclean_water_open: BOOL:= FALSE; //自洁喷杆球阀打开开路
	DO_Hpre_pump_short: BOOL:= FALSE; //高压水泵啮合短路
	DO_Hpre_pump_open: BOOL:= FALSE; //高压水泵啮合开路
	DO_fog_Spump_short: BOOL:= FALSE; //低压隔膜泵打开短路
	DO_fog_Spump_open: BOOL:= FALSE; //低压隔膜泵打开开路
	DO_Motor_en_short: BOOL:= FALSE; //电机使能控制短路
	DO_Motor_en_open: BOOL:= FALSE; //电机使能控制开路
	DO_watercooler_pump_short: BOOL:= FALSE; //水冷泵电机控制短路
	DO_watercooler_pump_open: BOOL:= FALSE; //水冷泵电机控制开路
	DO_cooler_fan_short: BOOL:= FALSE; //散热风扇控制短路
	DO_cooler_fan_open: BOOL:= FALSE; //散热风扇控制开路
	DO_backup_power_short: BOOL:= FALSE; //备用动力控制短路
	DO_backup_power_open: BOOL:= FALSE; //备用动力控制开路
	
	iccid :STRING;
	lac :UINT;
	cid :UINT;
	sn :STRING;
	work_time :UDINT;
	motor_work_time: DWORD;
	g_m26:fb_m26;
END_VAR

VAR_GLOBAL CONSTANT
	para_file:STRING:=ANY_TO_STRING("parameters.txt");
	gMagicNum :REAL := 12345.6789;   //magic number for check sum
END_VAR

// Changsha_Xiangji_ARM_Cortex_A9_xilinx_zynq7000_linux/Application/prg_main
PROGRAM prg_main  //主控制程序
VAR
	iStat:UINT:= 0;
	tmr_run:ton();
    bFirst		: BOOL 	:= TRUE ;
	bFirst1		: BOOL 	:= TRUE ;
	F_Motor_Work:F_TRIG;
	T_MotorSpd: Ton;
	T_DI_Totvalve_Open: Ton;
	T_DI_Totvalve_noOpen: Ton;
	// 高压水路球阀打开标志
	Totvalve_open_sign: BOOL;
	T_DI_Hpre_valve_open: Ton;
	T_DI_Hpre_valve_noOpen: Ton;
	// 吹净球阀打开标志
	Hpre_valve_sign: BOOL;

	// 全洗扫车上升沿
	R_HMI_AwashSweep: R_TRIG;
	// 工作模式限制
	work_mod_limit: BOOL;
	// 左洗扫上升沿
	R_HMI_LwashSweep: R_TRIG;
	// 右洗扫上升沿
	R_HMI_RwashSweep: R_TRIG;
	// 全扫路上升沿
	R_HMI_ASweeproad: R_TRIG;
	// 左扫路上升沿
	R_HMI_LSweeproad: R_TRIG;
	// 右扫路上升沿
	R_HMI_RSweeproad: R_TRIG;
	// 全清洗上升沿
	R_HMI_Aclean: R_TRIG;
	// 左清洗上升沿
	R_HMI_Lclean: R_TRIG;
	// 右清洗上升沿
	R_HMI_Rclean: R_TRIG;
	T_TEST_ALM: Ton;
	T_RCAR_ALM: Ton;
	T_Motor_Work_ALM: Ton;
	T_DI_Rcar_fault: TON;
	R_T_DI_Rcar: R_TRIG;
	R_Wastewater_full_Fault: R_TRIG;
	R_DI_Rcar_fault: R_TRIG;
	R_Wastewater_full_Fault1: R_TRIG;
	R_Chassis_SOC_LOW: R_TRIG;
	R_Sweep_stop: R_TRIG;
	T_Sweep_stop: TON;
	T_Lsweep_out1: Ton;

	T_DO_Lsweep_out1: Ton;
	T_DO_Lsweep_down1: Ton;

	T_Rsweep_out1: Ton;

	T_DO_Rsweep_out1: Ton;
	T_DO_Rsweep_down1: Ton;

	T_SYS_work: Ton;
	T_SYS_work1: Ton;

	// 左扫旋转中间变量1
	T_LSweep1: Ton;
	// 右扫旋转中间变量1
	T_RSweep1: Ton;

	// 右扫旋转中间变量下降沿
	F_T_RSweep1: F_TRIG;
	//全洗扫标志位上升沿
	R_AwashSweep_HMI: R_TRIG;
	//全扫路标志位上升沿
	R_ASweeproad_HMI: R_TRIG;
	// 右切全中间变量
	R_ASweep: BOOL;
	T_R_ASweep: TON;
	// 右洗扫标志位上升沿
	R_RwashSweep_HMI: R_TRIG;
	// 右扫路标志上升沿
	R_RSweeproad_HMI: R_TRIG;
	// 左扫旋转中间变量下降沿
	F_T_LSweep1: F_TRIG;
	// 左扫切全扫中间变量
	L_ASweep: BOOL;
	T_L_ASweep: TON;
	// 左洗扫标志位上升沿
	R_LwashSweep_HMI: R_TRIG;
	// 左扫路标志位上升沿
	R_LSweeproad_HMI: R_TRIG;
	// 全扫旋转标志位下降沿
	F_ASweep: F_TRIG;
	// 全扫切右扫中间变量
	A_RSweep: BOOL;
	T_A_RSweep: TON;
	// 全扫切左扫中间变量
	A_LSweep: BOOL;
	T_A_LSweep: Ton;
	// 左扫盘上升时间
	T_Lsweep_up: Ton;
	// 左扫盘上升标志位
	DO_Lsweep_up1: BOOL;
	T_Rsweep_up: Ton;

	T_Suction_Up: Ton;
	// 吸嘴球阀打开标志
	T_DO_Suction_water: Ton;
	// 左喷杆球阀打开标志
	T_DO_Lrod_water: Ton;

	// 右喷杆球阀打开标志位
	T_DO_Rrod_water: Ton;
	// 扫路延时标志位
	T_Sweeproad: Ton;
	// 喷雾降尘泵上升沿
	R_HMI_fog_Spump: R_TRIG;

	// 喷雾降尘泵中间变量
	DO_fog_Spump100: BOOL;
	T_fog_Spump_arm: Ton;
	R_T_Sweeproad: R_TRIG;
	F_T_Sweeproad: F_TRIG;
	R_Aclean_HMI: R_TRIG;
	R_Lclean_HMI: R_TRIG;
	R_Rclean_HMI: R_TRIG;
	R_HMI_wastewater_pump: R_TRIG;
	// 辅污水箱1满上升沿
	R_T_DI_auxiliary1_warte_H: R_TRIG;
	// 辅污水箱2满上升沿
	R_T_DI_auxiliary2_warte_H: R_TRIG;
	// 污水泵打开后延时10分钟
	T_DO_wastewater_pump_open1: Ton;
	// 自动排污上升沿
	R_auto_wastewater_pump: R_TRIG;
	// 污水泵工作10分钟后上升沿
	R_T_DO_wastewater_pump_open1: R_TRIG;
	// 污水泵打开中间变量
	DO_wastewater_pump_open100: BOOL;
	// 污水泵球阀打开标志位
	T_DO_wastewater_valve_open: Ton;
	// 高压水泵打开条件标志位
	Hpre_waterpump_open_pre: BOOL;

	// 高压冲洗上升沿
	R_HMI_Hpre_wash: R_TRIG;
	// 高压冲洗中间变量
	DO_Hpressure_water100: BOOL;
	// 功能测试上升沿
	R_Func_test_HMI: R_TRIG;
	// 高压水泵打开条件下降沿
	F_Hpre_waterpump_open_pre: F_TRIG;
	// 自洁上升沿
	R_HMI_selfclean: R_TRIG;

	// 自洁中间变量
	DO_selfclean_water100: BOOL;
	// 高压水泵提前启动寄存器
	Hpre_waterpump_open_pre1: BOOL;
	// 高压水泵打开中间变量
	Hpre_waterpump_open_Mid: BOOL;
	// 高压冲洗标志位上升沿
	R_DO_Hpressure_water1: R_TRIG;
	// 自洁标志位上升沿
	R_DO_selfclean_water1: R_TRIG;
	// 高压冲洗标志位下降沿
	F_DO_Hpressure_water1: F_TRIG;
	// 自洁标志位下降沿
	F_DO_selfclean_water1: F_TRIG;
	// 高压水泵打开中间变量上升沿
	R_Hpre_waterpump_open_Mid: R_TRIG;
	// 高压水泵啮合中间寄存器1
	Hpre_waterpump_open_Mid1: BOOL;
	// 高压水泵啮合中间寄存器2
	Hpre_waterpump_open_Mid2: BOOL;
	// 给定值暂存寄存器
	SETspeed_1: UINT;
	// 电机实际速度与给定速度偏差
	SETspeed_2: UINT;
	// 实际值与怠速偏差
	Speed_Dif: BOOL;
	T_Hpre_waterpump_open_Mid1: Ton;
	// 实际值与给定值偏差上升沿
	R_Speed_Dif: R_TRIG;
	R_T_Hpre_waterpump_open_Mid1: R_TRIG;
	T_Hpre_waterpump_open_Mid2: Ton;
	R_T_Hpre_waterpump_open_Mid2: R_TRIG;
	// M78下降沿
	F_Hpre_waterpump_open_Mid: F_TRIG;

	tmp_byte: INT;

	// 电机启动变量
	motor_start: BOOL;
	// 电机启动延时25S
	T_HMI_start_motor: Ton;
	// 电机启动中间变量
	motor_start_Mid: BOOL;
	// 电机开始启动定时器
	T_HMI_start_motor1: Ton;
	// 电机启动开始上升沿
	R_T_HMI_start_motor1: R_TRIG;
	// 停扫标志上升沿
	R_Sweep_stop_HMI: R_TRIG;
	// 启动超时
	HMI_start_motor_overT: BOOL;
	// 启动超时时间
	T_HMI_start_motor_overT: Ton;
	// 备用动力开关触发停机上升沿
	R_backup_power_stopmotor: R_TRIG;
	// 电机故障停机定时器
	T_motor_fault: Ton;

	// 水冷泵延时6S停机
	T_DO_watercooler_pump_open1: Ton;
	// 系统工作上升沿
	R_sys_work: R_TRIG;
	// 智能标志下降沿
	F_Intelligent_HMI: F_TRIG;
	// 标准工作转速上升沿
	R_HMI_Standard_speed: R_TRIG;
	// 强力工作速度上升沿
	R_HMI_Strong_speed: R_TRIG;
	// 电机减速上升沿
	R_HMI_Dec_Speed: R_TRIG;
	// 电机加速上升沿
	R_HMI_Inc_Speed: R_TRIG;
	// 高速上升沿
	R_HMI_Sweep_Hspd: R_TRIG;
	// 中速上升沿
	R_HMI_Sweep_Mspd: R_TRIG;
	// 低速上升沿
	R_HMI_Sweep_Lspd: R_TRIG;
	// 车辆停止
	T_Chassis_stop: Ton;
	// 车速低速
	T_Chassis_Lspeed: Ton;
	// 车辆中低速
	T_Chassis_M_Lspeed: Ton;
	// 车辆中高速
	T_Chassis_M_Hspeed: Ton;
	// 车辆高速
	T_Chassis_Hspeed: Ton;
	// 智能上升沿
	R_HMI_intelligent: R_TRIG;
	// 清洁上升沿
	R_HMI_cleanly: R_TRIG;
	// 一般上升沿
	R_HMI_normal: R_TRIG;
	// 污染上升沿
	R_HMI_dirty: R_TRIG;
	// 智能中间变量
	Intelligent_HMI100: BOOL;
	// 系统工作下降沿
	F_sys_work: F_TRIG;
	// 扫盘上升
	JX_sweep_up: BOOL;
	// 扫盘下降
	JX_Sweep_Down: BOOL;
	// 扫盘摆出
	JX_Sweep_out: BOOL;
	// 扫盘缩回
	JX_Sweep_return: BOOL;
	T_DI_oil_release_valve: Ton;
	// 检修盒备用动力打开
	JX_backup_power_open: BOOL;
	// 更换扫刷上升沿
	R_HMI_replace_Sweep: R_TRIG;
	// 更换扫刷中间变量
	replace_Sweep_HMI1: BOOL;
	T_HMI_MOTOR_runstop_M: TON;
	

	// 电驱CAN通讯失败上升沿
	R_T_Motor_CAN_fault: R_TRIG;
	// 冬季排水启动上升沿
	R_HMI_drain_start: R_TRIG;
	// 冬季排水启动中间变量
	Drain_start_HMI100: BOOL;
	// 冬季排水手动上升沿
	R_HMI_drain_manual: R_TRIG;
	R_HMI_drain_auto: R_TRIG;
	Drain_auto_HMI100: BOOL;
	// 左喷杆排水手动
	Lrod_drain_HMI_manu: BOOL;
	// 右喷杆排水手动
	Rrod_drain_HMI_manu: BOOL;
	// 吸嘴喷杆排水手动
	Suction_drain_HMI_manu: BOOL;
	// 高辅喷杆排水手动
	Hpressure_drain_HMI_manu: BOOL;
	// 自洁喷杆排水手动
	Selfclean_drain_HMI_manu: BOOL;
	// 左喷杆排水自动
	Lrod_drain_HMI_auto: BOOL;
	// 右喷杆排水自动
	Rrod_drain_HMI_auto: BOOL;
	// 吸嘴喷杆排水自动
	Suction_drain_HMI_auto: BOOL;
	// 高辅喷杆排水自动
	Hpressure_drain_HMI_auto: BOOL;
	// 自洁喷杆排水自动
	Selfclean_drain_HMI_auto: BOOL;
	T_Lrod_drain_HMI_auto: Ton;
	T_Rrod_drain_HMI_auto: Ton;
	T_Suction_drain_HMI_auto: Ton;
	T_Hpressure_drain_HMI_auto: Ton;
	T_Selfclean_drain_HMI_auto: Ton;
	i: BOOL := TRUE ;
	

	
	
	k: BOOL := FALSE;
	T_ASweep1: TON;
	R_Hpre_waterpump_open_Mid1: R_TRIG;
	R_T_fog_pump_press_noOk: R_TRIG;
	R_Intelligent_HMI: R_TRIG;
	count1: INT:=0;
	motor_stop: BOOL := FALSE;
	R_motor_stop: R_TRIG;
END_VAR

VAR CONSTANT

	
END_VAR


//初始化时读取参数，程序运行过程中直接使用g_parameters.para_val[i]访问参数； 
//如果修改了参数，则需要手动调用 fn_write_para_file(g_parameters)来保存到硬盘;
(*CASE iStat OF
	0: //init
		fn_read_para_file(ADR(g_parameters)); 
		
		
		IF NOT g_parameters.para_ok THEN  //读取参数失败，设置初始值
			g_parameters.para_val[0] := 50;//加减值
			g_parameters.para_val[1] := 850;//最低转速
			g_parameters.para_val[2] := 1450;//标准转速
			g_parameters.para_val[3] := 1750;//强力转速
			g_parameters.para_val[4] := 0;//扫盘转速
			g_parameters.para_val[5] := 1850;//高压水泵超速报警
			g_parameters.para_val[6] := 1950;//高压水泵超速停止
			g_parameters.para_val[7] := 2500;//最高转速
			g_parameters.para_val[8] := 850;//怠速
			g_parameters.para_val[9] := 1000;//清洁低速
			g_parameters.para_val[10] := 1000;//清洁中低速
			g_parameters.para_val[11] := 1100;//清洁中高速
			g_parameters.para_val[12] := 1450;//清洁高速
			g_parameters.para_val[13] := 1200;//一般低速
			g_parameters.para_val[14] := 1350;//一般中低速
			g_parameters.para_val[15] := 1500;//一般中高速
			g_parameters.para_val[16] := 1750;//一般高速
			g_parameters.para_val[17] := 1350;//污染低速
			g_parameters.para_val[18] := 1550;//污染中低速
			g_parameters.para_val[19] := 1750;//污染中高速
			g_parameters.para_val[20] := 1750;//污染高速
			g_parameters.para_val[21] := 100;
			g_parameters.para_ok := TRUE;
			fn_write_para_file(g_parameters);
			ELSE
			S_IncDec_Speed:=ANY_TO_UINT(g_parameters.para_val[0]); 
				
		END_IF
		
		iSTat := 10;

	10:
	
END_CASE
*)
tmr_run(in := TRUE, pt := TIME#500MS);
IF tmr_run.Q THEN
	%QX156.0 := NOT %QX156.0; 
	tmr_run(in := FALSE);
END_IF
(*
//********设置参数例子
IF Re_IncDec_Speed>0 AND S_IncDec_Speed<>Re_IncDec_Speed THEN
	g_parameters.para_val[0] := Re_IncDec_Speed;//加减值
	fn_write_para_file(g_parameters);
    S_IncDec_Speed :=Re_IncDec_Speed;   
END_IF
*)
//调用读写falsh
FALSH_RW();
//调用DO输出故障判断
//DO_fault();

//电机工作时间
IF motor_work THEN
	count1:=count1+1;
END_IF
IF count1=1200 THEN
	motor_work_time :=motor_work_time+1;
	count1:=0;
	g_parameters.para_val[22] :=ANY_TO_UINT(motor_work_time MOD 256);
	g_parameters.para_val[23] :=ANY_TO_UINT(motor_work_time/16#100);
	g_parameters.para_val[24] :=ANY_TO_UINT(motor_work_time/16#10000);
	g_parameters.para_val[25] :=ANY_TO_UINT(motor_work_time/16#1000000);
	fn_write_para_file(g_parameters);
END_IF


//功能测试调用
Func_test_HMI:=HMI_func_test;(* 功能测试标志*)
IF Func_test_HMI AND (NOT SYS_work) THEN
    TEST();
END_IF
//功能测试参数初始化
IF bFirst OR (NOT Func_test_HMI)  THEN
    bFirst := FALSE ;
   	cooler_motor_Test:=FALSE;
	cooler_fan_Test:=FALSE;
	Sweep_Mspeed_Test:=FALSE;
    Sweep_Lspeed_Test:=FALSE;
	LSweep_Test:=FALSE;
    RSweep_Test:=FALSE;
    ASweep_Test:=FALSE;
	LSweep_out_Test:=FALSE;
	RSweep_out_Test:=FALSE;
	Lrod_OUT_Test:=FALSE;
	Rrod_OUT_Test:=FALSE;
	Lrod_water_Test:=FALSE;
	Rrod_water_Test:=FALSE;
	Suction_water_Test:=FALSE;
	Hpre_wash_Test:=FALSE;
	selfclean_water_Test:=FALSE;
	Hpress_pump_gearin_Test:=FALSE;
	Fog_pump_Test:=FALSE;
	Wastewater_pump_Test:=FALSE;
	Wastewater_valve_Test:=FALSE;
	Backup_power_Test:=FALSE;
END_IF

//参数初始化
F_Motor_Work(CLK:=Motor_Work);
IF bFirst1 OR F_Motor_Work.Q THEN
    bFirst1 := FALSE ;
    Sweep_HSpeed_HMI:=(S_Sweep_Speed =0);(* 扫盘高速 *)
    Sweep_MSpeed_HMI:=(S_Sweep_Speed =1);(* 扫盘中速 *)
    Sweep_LSpeed_HMI:=(S_Sweep_Speed =2);(* 扫盘低速 *)
	
END_IF

//发动机工作判断 
T_MotorSpd(IN:=Motor_real_speed_HMI>250,PT:=T#2S);
IF T_MotorSpd.Q THEN
     Motor_Work:=TRUE;
ELSE
     Motor_Work:=FALSE;
END_IF

//高压水路球阀位置判断
T_DI_Totvalve_Open(IN:=DI_Totvalve_Open,PT:=T#1S);
T_DI_Totvalve_noOpen(IN:=(NOT DI_Totvalve_Open),PT:=T#1S);
IF T_DI_Totvalve_Open.Q  THEN
      Totvalve_open_sign:=TRUE;
ELSIF T_DI_Totvalve_noOpen.Q THEN
	  Totvalve_open_sign:=FALSE;  
END_IF
//高压吹净球阀位置判断
T_DI_Hpre_valve_Open(IN:=DI_Hpre_valve_Open,PT:=T#1S);
T_DI_Hpre_valve_noOpen(IN:=(NOT DI_Hpre_valve_Open),PT:=T#1S);
IF T_DI_Hpre_valve_Open.Q  THEN
      Hpre_valve_sign:=TRUE;
ELSIF T_DI_Hpre_valve_noOpen.Q THEN
	  Hpre_valve_sign:=FALSE;  
END_IF
//水路卸荷阀故障判断
T_water_overflow_noClose(IN:=(NOT DO_water_overflow) AND (NOT DI_water_overflow),PT:=T#7S);(*水路卸荷发未关闭故障*)
T_water_overflow_noOpen(IN:=DO_water_overflow AND DI_water_overflow,PT:=T#7S);(*水路卸荷阀未打开故障*)
//喷雾降尘泵压力判断
T_fog_pump_press_noOk(IN:=NOT DI_fog_pump_press_ok,PT:=T#10S);(*喷雾降尘泵压力不正常*)
//主污水箱水满判断
T_DI_wastewater_full(IN:=DI_wastewater_full,PT:=T#6S);(*主污水箱水满标志*)
//辅污水箱1水满判断
T_DI_auxiliary1_warte_H(IN:=DI_auxiliary1_warte_H,PT:=T#6S);(*辅污水箱1水满标志*)
//辅污水箱2水满判断
T_DI_auxiliary2_warte_H(IN:=DI_auxiliary2_warte_H,PT:=T#6S);(*辅污水箱2水满标志*)
//污水满判断
Wastewater_full_Fault:=T_DI_wastewater_full.Q AND (T_DI_auxiliary1_warte_H.Q OR T_DI_auxiliary2_warte_H.Q);
//辅助水箱水位不一致判断
T_auxiliary_warte_dif(IN:=((NOT T_DI_auxiliary2_warte_H.Q) AND T_DI_auxiliary1_warte_H.Q) OR ((NOT T_DI_auxiliary1_warte_H.Q) AND T_DI_auxiliary2_warte_H.Q),PT:=T#6S);
//回油过滤堵塞判断
T_DI_oil_filter_block(IN:=DI_oil_filter_block,PT:=T#6S);
//液压油位低判断
T_DI_oil_level_low(IN:=DI_oil_level_low,PT:=T#6S);
//气路系统压力判断
T_DI_air_press_low(IN:=DI_air_press_low,PT:=T#2S);
//倒车判断
T_DI_Rcar(IN:=DI_Rcar,PT:=T#2S);
//水箱水位低判断
T_DI_cleanwater_LOW(IN:=(DI_cleanwater_LOW>2500),PT:=T#5S);

//高压水泵超速报警
T_Pumpspeed_H(IN:=((Motor_real_speed_HMI>S_Pumpspeed_arm) AND DO_Hpre_pump1),PT:=T#5S);
//高压水泵超速停止
T_Pumpspeed_HH(IN:=((Motor_real_speed_HMI>S_Pumpspeed_stop) AND DO_Hpre_pump1),PT:=T#5S);

//工作模式限定条件 
work_mod_limit:=(NOT Func_test_HMI) AND Motor_Work AND (NOT T_DI_Rcar.Q);
//工作模式选择
//全洗扫模式
R_HMI_AwashSweep(CLK:=HMI_AwashSweep AND (NOT HMI_LwashSweep) AND (NOT HMI_RwashSweep) AND (NOT HMI_LSweeproad) AND (NOT HMI_ASweeproad)AND (NOT HMI_RSweeproad) AND (NOT HMI_Lcleanwash) AND (NOT HMI_Acleanwash) AND (NOT HMI_Rcleanwash) AND (NOT HMI_stop_sweep));
IF R_HMI_AwashSweep.Q AND work_mod_limit THEN
   AwashSweep_HMI:=TRUE;(* 全洗扫 *)
   LwashSweep_HMI:=FALSE;(* 左洗扫 *)
   RwashSweep_HMI:=FALSE;(* 右洗扫 *)
   ASweeproad_HMI:=FALSE;(* 全扫路 *)
   LSweeproad_HMI:=FALSE;(* 左扫路 *)
   RSweeproad_HMI:=FALSE;(* 右扫路 *)
   Aclean_HMI:=FALSE;(* 全清洗 *)
   Lclean_HMI:=FALSE;(* 左清洗 *)
   Rclean_HMI:=FALSE;(* 右清洗 *)
   Sweep_stop_HMI:=FALSE;(* 停扫 *)
END_IF
//左洗扫模式
R_HMI_LwashSweep(CLK:=(NOT HMI_AwashSweep) AND HMI_LwashSweep AND (NOT HMI_RwashSweep) AND (NOT HMI_LSweeproad) AND (NOT HMI_ASweeproad)AND (NOT HMI_RSweeproad) AND (NOT HMI_Lcleanwash) AND (NOT HMI_Acleanwash) AND (NOT HMI_Rcleanwash) AND (NOT HMI_stop_sweep));
IF R_HMI_LwashSweep.Q AND work_mod_limit THEN
   AwashSweep_HMI:=FALSE;(* 全洗扫 *)
   LwashSweep_HMI:=TRUE;(* 左洗扫 *)
   RwashSweep_HMI:=FALSE;(* 右洗扫 *)
   ASweeproad_HMI:=FALSE;(* 全扫路 *)
   LSweeproad_HMI:=FALSE;(* 左扫路 *)
   RSweeproad_HMI:=FALSE;(* 右扫路 *)
   Aclean_HMI:=FALSE;(* 全清洗 *)
   Lclean_HMI:=FALSE;(* 左清洗 *)
   Rclean_HMI:=FALSE;(* 右清洗 *)
   Sweep_stop_HMI:=FALSE;(* 停扫 *)
END_IF
//右洗扫模式
R_HMI_RwashSweep(CLK:=(NOT HMI_AwashSweep) AND (NOT HMI_LwashSweep) AND HMI_RwashSweep AND (NOT HMI_LSweeproad) AND (NOT HMI_ASweeproad)AND (NOT HMI_RSweeproad) AND (NOT HMI_Lcleanwash) AND (NOT HMI_Acleanwash) AND (NOT HMI_Rcleanwash) AND (NOT HMI_stop_sweep));
IF R_HMI_RwashSweep.Q AND work_mod_limit THEN
   AwashSweep_HMI:=FALSE;(* 全洗扫 *)
   LwashSweep_HMI:=FALSE;(* 左洗扫 *)
   RwashSweep_HMI:=TRUE;(* 右洗扫 *)
   ASweeproad_HMI:=FALSE;(* 全扫路 *)
   LSweeproad_HMI:=FALSE;(* 左扫路 *)
   RSweeproad_HMI:=FALSE;(* 右扫路 *)
   Aclean_HMI:=FALSE;(* 全清洗 *)
   Lclean_HMI:=FALSE;(* 左清洗 *)
   Rclean_HMI:=FALSE;(* 右清洗 *)
   Sweep_stop_HMI:=FALSE;(* 停扫 *)
END_IF
//全扫路模式
R_HMI_ASweeproad(CLK:=(NOT HMI_AwashSweep) AND (NOT HMI_LwashSweep) AND (NOT HMI_RwashSweep) AND (NOT HMI_LSweeproad) AND HMI_ASweeproad AND (NOT HMI_RSweeproad) AND (NOT HMI_Lcleanwash) AND (NOT HMI_Acleanwash) AND (NOT HMI_Rcleanwash) AND (NOT HMI_stop_sweep));
IF R_HMI_ASweeproad.Q AND work_mod_limit THEN
   AwashSweep_HMI:=FALSE;(* 全洗扫 *)
   LwashSweep_HMI:=FALSE;(* 左洗扫 *)
   RwashSweep_HMI:=FALSE;(* 右洗扫 *)
   ASweeproad_HMI:=TRUE;(* 全扫路 *)
   LSweeproad_HMI:=FALSE;(* 左扫路 *)
   RSweeproad_HMI:=FALSE;(* 右扫路 *)
   Aclean_HMI:=FALSE;(* 全清洗 *)
   Lclean_HMI:=FALSE;(* 左清洗 *)
   Rclean_HMI:=FALSE;(* 右清洗 *)
   Sweep_stop_HMI:=FALSE;(* 停扫 *)
END_IF
//左扫路模式
R_HMI_LSweeproad(CLK:=(NOT HMI_AwashSweep) AND (NOT HMI_LwashSweep) AND (NOT HMI_RwashSweep) AND HMI_LSweeproad AND (NOT HMI_ASweeproad)AND (NOT HMI_RSweeproad) AND (NOT HMI_Lcleanwash) AND (NOT HMI_Acleanwash) AND (NOT HMI_Rcleanwash) AND (NOT HMI_stop_sweep));
IF R_HMI_LSweeproad.Q AND work_mod_limit THEN
   AwashSweep_HMI:=FALSE;(* 全洗扫 *)
   LwashSweep_HMI:=FALSE;(* 左洗扫 *)
   RwashSweep_HMI:=FALSE;(* 右洗扫 *)
   ASweeproad_HMI:=FALSE;(* 全扫路 *)
   LSweeproad_HMI:=TRUE;(* 左扫路 *)
   RSweeproad_HMI:=FALSE;(* 右扫路 *)
   Aclean_HMI:=FALSE;(* 全清洗 *)
   Lclean_HMI:=FALSE;(* 左清洗 *)
   Rclean_HMI:=FALSE;(* 右清洗 *)
   Sweep_stop_HMI:=FALSE;(* 停扫 *)
END_IF
//右扫路模式
R_HMI_RSweeproad(CLK:=(NOT HMI_AwashSweep) AND (NOT HMI_LwashSweep) AND (NOT HMI_RwashSweep) AND (NOT HMI_LSweeproad) AND (NOT HMI_ASweeproad)AND HMI_RSweeproad AND (NOT HMI_Lcleanwash) AND (NOT HMI_Acleanwash) AND (NOT HMI_Rcleanwash) AND (NOT HMI_stop_sweep));
IF R_HMI_RSweeproad.Q AND work_mod_limit THEN
   AwashSweep_HMI:=FALSE;(* 全洗扫 *)
   LwashSweep_HMI:=FALSE;(* 左洗扫 *)
   RwashSweep_HMI:=FALSE;(* 右洗扫 *)
   ASweeproad_HMI:=FALSE;(* 全扫路 *)
   LSweeproad_HMI:=FALSE;(* 左扫路 *)
   RSweeproad_HMI:=TRUE;(* 右扫路 *)
   Aclean_HMI:=FALSE;(* 全清洗 *)
   Lclean_HMI:=FALSE;(* 左清洗 *)
   Rclean_HMI:=FALSE;(* 右清洗 *)
   Sweep_stop_HMI:=FALSE;(* 停扫 *)
END_IF
//全清洗模式
R_HMI_Aclean(CLK:=(NOT HMI_AwashSweep) AND (NOT HMI_LwashSweep) AND (NOT HMI_RwashSweep) AND (NOT HMI_LSweeproad) AND (NOT HMI_ASweeproad)AND (NOT HMI_RSweeproad) AND (NOT HMI_Lcleanwash) AND HMI_Acleanwash AND (NOT HMI_Rcleanwash) AND (NOT HMI_stop_sweep));
IF R_HMI_Aclean.Q AND work_mod_limit THEN
   AwashSweep_HMI:=FALSE;(* 全洗扫 *)
   LwashSweep_HMI:=FALSE;(* 左洗扫 *)
   RwashSweep_HMI:=FALSE;(* 右洗扫 *)
   ASweeproad_HMI:=FALSE;(* 全扫路 *)
   LSweeproad_HMI:=FALSE;(* 左扫路 *)
   RSweeproad_HMI:=FALSE;(* 右扫路 *)
   Aclean_HMI:=TRUE;(* 全清洗 *)
   Lclean_HMI:=FALSE;(* 左清洗 *)
   Rclean_HMI:=FALSE;(* 右清洗 *)
   Sweep_stop_HMI:=FALSE;(* 停扫 *)
END_IF
//左清洗模式
R_HMI_Lclean(CLK:=(NOT HMI_AwashSweep) AND (NOT HMI_LwashSweep) AND (NOT HMI_RwashSweep) AND (NOT HMI_LSweeproad) AND (NOT HMI_ASweeproad)AND (NOT HMI_RSweeproad) AND HMI_Lcleanwash AND (NOT HMI_Acleanwash) AND (NOT HMI_Rcleanwash) AND (NOT HMI_stop_sweep));
IF R_HMI_Lclean.Q AND work_mod_limit THEN
   AwashSweep_HMI:=FALSE;(* 全洗扫 *)
   LwashSweep_HMI:=FALSE;(* 左洗扫 *)
   RwashSweep_HMI:=FALSE;(* 右洗扫 *)
   ASweeproad_HMI:=FALSE;(* 全扫路 *)
   LSweeproad_HMI:=FALSE;(* 左扫路 *)
   RSweeproad_HMI:=FALSE;(* 右扫路 *)
   Aclean_HMI:=FALSE;(* 全清洗 *)
   Lclean_HMI:=TRUE;(* 左清洗 *)
   Rclean_HMI:=FALSE;(* 右清洗 *)
   Sweep_stop_HMI:=FALSE;(* 停扫 *)
END_IF
//右清洗模式
R_HMI_Rclean(CLK:=(NOT HMI_AwashSweep) AND (NOT HMI_LwashSweep) AND (NOT HMI_RwashSweep) AND (NOT HMI_LSweeproad) AND (NOT HMI_ASweeproad)AND (NOT HMI_RSweeproad) AND (NOT HMI_Lcleanwash) AND (NOT HMI_Acleanwash) AND HMI_Rcleanwash AND (NOT HMI_stop_sweep));
IF R_HMI_Rclean.Q AND work_mod_limit THEN
   AwashSweep_HMI:=FALSE;(* 全洗扫 *)
   LwashSweep_HMI:=FALSE;(* 左洗扫 *)
   RwashSweep_HMI:=FALSE;(* 右洗扫 *)
   ASweeproad_HMI:=FALSE;(* 全扫路 *)
   LSweeproad_HMI:=FALSE;(* 左扫路 *)
   RSweeproad_HMI:=FALSE;(* 右扫路 *)
   Aclean_HMI:=FALSE;(* 全清洗 *)
   Lclean_HMI:=FALSE;(* 左清洗 *)
   Rclean_HMI:=TRUE;(* 右清洗 *)
   Sweep_stop_HMI:=FALSE;(* 停扫 *)
END_IF
//请关闭测试提示
IF Func_test_HMI AND (R_HMI_AwashSweep.Q OR R_HMI_LwashSweep.Q OR R_HMI_RwashSweep.Q OR R_HMI_ASweeproad.Q OR R_HMI_LSweeproad.Q OR R_HMI_RSweeproad.Q OR R_HMI_Aclean.Q OR R_HMI_Lclean.Q OR R_HMI_Rclean.Q) THEN
   TEST_ALM:=TRUE;(* 工作操作时，请关闭测试提示标志位 *)
   ELSIF T_TEST_ALM.Q THEN
   TEST_ALM:=FALSE;
END_IF
T_TEST_ALM(IN:=TEST_ALM,PT:=T#1.0S);
//倒车提示
IF T_DI_Rcar.Q AND (R_HMI_AwashSweep.Q OR R_HMI_LwashSweep.Q OR R_HMI_RwashSweep.Q OR R_HMI_ASweeproad.Q OR R_HMI_LSweeproad.Q OR R_HMI_RSweeproad.Q OR R_HMI_Aclean.Q OR R_HMI_Lclean.Q OR R_HMI_Rclean.Q) THEN
   RCAR_ALM:=TRUE;(* 正在倒车中提示 *)
   ELSIF T_TEST_ALM.Q THEN
   RCAR_ALM:=FALSE;
END_IF
T_RCAR_ALM(IN:=RCAR_ALM,PT:=T#1.0S);
//请先打开发动机
IF (NOT Motor_work) AND (R_HMI_AwashSweep.Q OR R_HMI_LwashSweep.Q OR R_HMI_RwashSweep.Q OR R_HMI_ASweeproad.Q OR R_HMI_LSweeproad.Q OR R_HMI_RSweeproad.Q OR R_HMI_Aclean.Q OR R_HMI_Lclean.Q OR R_HMI_Rclean.Q) THEN
   Motor_Work_ALM:=TRUE;(* 请先打开电机 *)
   ELSIF T_Motor_Work_ALM.Q THEN
   Motor_Work_ALM:=FALSE;
END_IF
T_Motor_Work_ALM(IN:=Motor_Work_ALM,PT:=T#1.0S);
//倒车故障停机
T_DI_Rcar_fault(IN:=DI_Rcar_fault ,PT:=T#1.0S);
R_T_DI_Rcar(CLK:=T_DI_Rcar.Q);
IF R_T_DI_Rcar.Q AND SYS_work THEN
   DI_Rcar_fault:=TRUE;(* 倒车故障停机 *)
   ELSIF T_DI_Rcar_fault.Q THEN
   DI_Rcar_fault:=FALSE;
END_IF
//污水满故障停机
T_DI_Rcar_fault(IN:=DI_Rcar_fault ,PT:=T#1.0S);
R_Wastewater_full_Fault(CLK:=Wastewater_full_Fault);
IF R_Wastewater_full_Fault.Q AND SYS_work THEN
   Wastewater_full_Fault1:=TRUE;(* 污水满故障停机 *)
   ELSIF T_DI_Rcar_fault.Q THEN
   Wastewater_full_Fault1:=FALSE;
END_IF
//故障停机
Fault_STOP:=DI_Rcar_fault OR Wastewater_full_Fault1;
R_DI_Rcar_fault(CLK:=DI_Rcar_fault);
R_Wastewater_full_Fault1(CLK:=Wastewater_full_Fault1);
R_Chassis_SOC_LOW(CLK:=Chassis_SOC_LOW);
R_Sweep_stop(CLK:=HMI_stop_sweep);
IF R_DI_Rcar_fault.Q OR R_Wastewater_full_Fault1.Q OR (R_Chassis_SOC_LOW.Q AND SYS_work) OR R_Sweep_stop.Q OR HMI_MOTOR_runstop_M THEN
   AwashSweep_HMI:=FALSE;(* 全洗扫 *)
   LwashSweep_HMI:=FALSE;(* 左洗扫 *)
   RwashSweep_HMI:=FALSE;(* 右洗扫 *)
   ASweeproad_HMI:=FALSE;(* 全扫路 *)
   LSweeproad_HMI:=FALSE;(* 左扫路 *)
   RSweeproad_HMI:=FALSE;(* 右扫路 *)
   Aclean_HMI:=FALSE;(* 全清洗 *)
   Lclean_HMI:=FALSE;(* 左清洗 *)
   Rclean_HMI:=FALSE;(* 右清洗 *)
   Sweep_stop_HMI:=TRUE;(* 停扫 *)
   Intelligent_HMI:=FALSE;(* 智能 *)
  
END_IF
T_Sweep_stop(IN:=Sweep_stop_HMI,PT:=T#14S);(* 停扫14S后自动复位 *)
IF T_Sweep_stop.Q THEN
   Sweep_stop_HMI:=FALSE;
END_IF
//系统工作
SYS_work:=(AwashSweep_HMI OR LwashSweep_HMI OR RwashSweep_HMI OR ASweeproad_HMI OR LSweeproad_HMI OR RSweeproad_HMI OR Aclean_HMI OR Lclean_HMI OR Rclean_HMI);
//左扫盘摆出控制
T_Lsweep_out1(IN:=NOT (AwashSweep_HMI OR LwashSweep_HMI OR ASweeproad_HMI OR LSweeproad_HMI),PT:=T#3S);
IF AwashSweep_HMI OR LwashSweep_HMI OR ASweeproad_HMI OR LSweeproad_HMI THEN
    DO_Lsweep_out1:=TRUE;
ELSIF T_Lsweep_out1.Q THEN
    DO_Lsweep_out1:=FALSE;	
END_IF
//左扫盘摆出5S后下降
T_DO_Lsweep_out1(IN:=AwashSweep_HMI OR LwashSweep_HMI OR ASweeproad_HMI OR LSweeproad_HMI,PT:=T#5S);
T_DO_Lsweep_down1(IN:=T_DO_Lsweep_out1.Q,PT:=T#5S);
DO_Lsweep_down1:=T_DO_Lsweep_out1.Q AND (NOT T_DO_Lsweep_down1.Q)  ;
//右扫盘摆出控制
T_Rsweep_out1(IN:=NOT (AwashSweep_HMI OR RwashSweep_HMI OR ASweeproad_HMI OR RSweeproad_HMI),PT:=T#3S);
IF AwashSweep_HMI OR RwashSweep_HMI OR ASweeproad_HMI OR RSweeproad_HMI THEN
    DO_Rsweep_out1:=TRUE;
ELSIF T_Rsweep_out1.Q THEN
    DO_Rsweep_out1:=FALSE;	
END_IF
//右扫盘摆出后5S后下降
T_DO_Rsweep_out1(IN:=AwashSweep_HMI OR RwashSweep_HMI OR ASweeproad_HMI OR RSweeproad_HMI,PT:=T#5S);
T_DO_Rsweep_down1(IN:=T_DO_Rsweep_out1.Q,PT:=T#5S);
DO_Rsweep_down1:=T_DO_Rsweep_out1.Q AND (NOT T_DO_Rsweep_down1.Q);
//吸盘下降
T_SYS_work(IN:=SYS_work,PT:=T#7S);
T_SYS_work1(IN:=SYS_work,PT:=T#14S);
DO_Suction_Down1:=T_SYS_work.Q AND (NOT T_SYS_work1.Q);
//系统启动12S后扫旋转
T_LSweep1(IN:=LwashSweep_HMI OR LSweeproad_HMI,PT:=T#10S);(*左扫旋转中间变量*)
T_RSweep1(IN:=RwashSweep_HMI OR RSweeproad_HMI,PT:=T#10S);(*右扫旋转中间变量*)
T_ASweep1(IN:=AwashSweep_HMI OR ASweeproad_HMI,PT:=T#10S);
ASweep:=T_ASweep1.Q AND (NOT LSweep) AND (NOT RSweep);(*全扫旋转标志*)
//右扫切全扫控制
F_T_RSweep1(CLK:=T_RSweep1.Q);//右扫旋转中间变量下降沿
R_AwashSweep_HMI(CLK:=AwashSweep_HMI);//全洗扫标志位上升沿
R_ASweeproad_HMI(CLK:=ASweeproad_HMI);//全扫路标志位上升沿
T_R_ASweep(IN:=R_ASweep AND ((NOT R_RwashSweep_HMI.Q) OR (NOT R_RSweeproad_HMI.Q)),PT:=T#12S);
IF F_T_RSweep1.Q AND (R_AwashSweep_HMI.Q OR R_ASweeproad_HMI.Q) AND (NOT LwashSweep_HMI) AND (NOT LSweeproad_HMI) AND(NOT Aclean_HMI) AND(NOT Lclean_HMI) AND(NOT Rclean_HMI) AND(NOT Sweep_stop_HMI) THEN
	R_ASweep:=TRUE;//右扫切全扫中间变量
ELSIF T_R_ASweep.Q OR LwashSweep_HMI OR LSweeproad_HMI OR Aclean_HMI OR Lclean_HMI OR Rclean_HMI OR Sweep_stop_HMI THEN
	R_ASweep:=FALSE;//右扫切全扫中间变量
END_IF
R_RwashSweep_HMI(CLK:=RwashSweep_HMI);//右洗扫标志位上升沿
R_RSweeproad_HMI(CLK:=RSweeproad_HMI);//右洗扫标志位上升沿
//左扫切全扫控制
F_T_LSweep1(CLK:=T_LSweep1.Q);//左扫旋转中间变量下降沿
T_L_ASweep(IN:=L_ASweep AND ((NOT R_LwashSweep_HMI.Q) OR (NOT R_LSweeproad_HMI.Q)),PT:=T#12S);
IF F_T_LSweep1.Q AND (R_AwashSweep_HMI.Q OR R_ASweeproad_HMI.Q) AND (NOT RwashSweep_HMI) AND (NOT RSweeproad_HMI) AND(NOT Aclean_HMI) AND(NOT Lclean_HMI) AND(NOT Rclean_HMI) AND(NOT Sweep_stop_HMI) THEN 
	L_ASweep:=TRUE;//左扫切全扫中间变量
ELSIF T_L_ASweep.Q OR RwashSweep_HMI OR RSweeproad_HMI OR Aclean_HMI OR Lclean_HMI OR Rclean_HMI OR Sweep_stop_HMI THEN
	L_ASweep:=FALSE;//左扫切全扫中间变量		
END_IF
R_LwashSweep_HMI(CLK:=LwashSweep_HMI);//左洗扫标志位上升沿
R_LSweeproad_HMI(CLK:=LSweeproad_HMI);//左扫路标志位上升沿
//全扫切右扫控制
F_ASweep(CLK:=ASweep);//全扫旋转标志位下降沿
T_A_RSweep(IN:=A_RSweep AND ((NOT R_AwashSweep_HMI.Q) OR (NOT R_ASweeproad_HMI.Q)),PT:=T#12S);
IF F_ASweep.Q AND (R_RwashSweep_HMI.Q OR R_RSweeproad_HMI.Q) AND (NOT LwashSweep_HMI) AND (NOT LSweeproad_HMI) AND (NOT Aclean_HMI) AND (NOT Lclean_HMI) AND (NOT Rclean_HMI) AND (NOT Sweep_stop_HMI) THEN
	A_RSweep:=TRUE;//全扫切右扫中间变量
ELSIF T_A_RSweep.Q OR LwashSweep_HMI OR LSweeproad_HMI OR Aclean_HMI OR Lclean_HMI OR Rclean_HMI OR Sweep_stop_HMI THEN 
	A_RSweep:=FALSE;//全扫切右扫中间变量
END_IF
//全扫切左扫控制
T_A_LSweep(IN:=A_LSweep AND ((NOT R_AwashSweep_HMI.Q) OR (NOT R_ASweeproad_HMI.Q)),PT:=T#12S);
IF F_ASweep.Q AND (R_LwashSweep_HMI.Q OR R_LSweeproad_HMI.Q) AND (NOT  RwashSweep_HMI) AND (NOT  RSweeproad_HMI) AND (NOT  Aclean_HMI) AND (NOT  Lclean_HMI) AND (NOT  Rclean_HMI) AND (NOT  Sweep_stop_HMI) THEN
    A_LSweep:=TRUE;//全扫切左扫中间变量
ELSIF T_A_LSweep.Q OR RwashSweep_HMI OR RSweeproad_HMI OR Aclean_HMI OR Lclean_HMI OR Rclean_HMI OR Sweep_stop_HMI THEN
	A_LSweep:=FALSE;//全扫切左扫中间变量
END_IF
//左扫旋转
LSweep:=(T_LSweep1.Q OR L_ASweep OR A_LSweep) AND (NOT ASweep) AND (NOT RSweep);
//右扫旋转
RSweep:=(T_RSweep1.Q OR R_ASweep OR A_RSweep) AND (NOT ASweep) AND (NOT LSweep);
//左扫盘上升
T_Lsweep_up(IN:=RwashSweep_HMI AND RSweeproad_HMI AND Sweep_stop_HMI AND Aclean_HMI AND Lclean_HMI AND Rclean_HMI,PT:=T#5S);
DO_Lsweep_up1:=(NOT T_Lsweep_up.Q) AND(RwashSweep_HMI OR RSweeproad_HMI OR Sweep_stop_HMI OR Aclean_HMI OR Lclean_HMI OR Rclean_HMI); 
//右扫盘上升
T_Rsweep_up(IN:=LwashSweep_HMI AND LSweeproad_HMI AND Sweep_stop_HMI AND Aclean_HMI AND Lclean_HMI AND Rclean_HMI,PT:=T#5S);
DO_Rsweep_up1:=(NOT T_Rsweep_up.Q) AND(LwashSweep_HMI OR LSweeproad_HMI OR Sweep_stop_HMI OR Aclean_HMI OR Lclean_HMI OR Rclean_HMI); 
//吸盘上升
T_Suction_Up(IN:=Sweep_stop_HMI,PT:=T#7S);
DO_Suction_Up1:=(NOT T_Suction_Up.Q) AND Sweep_stop_HMI;
//吸盘喷杆球阀控制
T_DO_Suction_water(IN:=AwashSweep_HMI OR LwashSweep_HMI OR RwashSweep_HMI OR Aclean_HMI OR Rclean_HMI OR Lclean_HMI,PT:=T#7S);
//左喷杆摆出、左喷杆球阀打开
DO_Lrod_out1:=AwashSweep_HMI OR LwashSweep_HMI OR Aclean_HMI OR Lclean_HMI;
T_DO_Lrod_water(IN:=AwashSweep_HMI OR LwashSweep_HMI OR Aclean_HMI OR Lclean_HMI,PT:=T#7S);
//右喷杆摆出、右喷杆球阀打开
DO_Rrod_out1:=AwashSweep_HMI OR RwashSweep_HMI OR Aclean_HMI OR Rclean_HMI;
T_DO_Rrod_water(IN:=AwashSweep_HMI OR RwashSweep_HMI OR Aclean_HMI OR Rclean_HMI,PT:=T#7S);
//低压隔膜泵控制
T_Sweeproad(IN:=ASweeproad_HMI OR LSweeproad_HMI OR RSweeproad_HMI,PT:=T#7S);
R_T_Sweeproad(CLK:=T_Sweeproad.Q);
F_T_Sweeproad(CLK:=T_Sweeproad.Q);
R_HMI_fog_Spump(CLK:=HMI_fog_Spump);
R_Aclean_HMI(CLK:=Aclean_HMI);
R_Lclean_HMI(CLK:=Lclean_HMI);
R_Rclean_HMI(CLK:=Rclean_HMI);
IF ((R_HMI_fog_Spump.Q AND (NOT DO_fog_Spump100)) OR R_T_Sweeproad.Q) AND Totvalve_open_sign AND (NOT T_DI_cleanwater_LOW.Q) AND DI_fog_pump_press_ok THEN
	DO_fog_Spump1:=TRUE;
ELSIF ((NOT Totvalve_open_sign)OR T_DI_cleanwater_LOW.Q OR R_HMI_fog_Spump.Q OR F_T_Sweeproad.Q OR R_Aclean_HMI.Q OR R_Lclean_HMI.Q OR R_Rclean_HMI.Q) AND DO_fog_Spump100 THEN
	DO_fog_Spump1:=FALSE;
END_IF
DO_fog_Spump100:=DO_fog_Spump1;
//隔膜泵球阀未打开
R_T_fog_pump_press_noOk(CLK:=T_fog_pump_press_noOk.Q);
T_fog_Spump_arm(IN:=fog_Spump_arm,PT:=T#1S);
IF R_T_fog_pump_press_noOk.Q AND DO_fog_Spump1 THEN
	fog_Spump_arm:=TRUE;
ELSIF T_fog_Spump_arm.Q THEN
	fog_Spump_arm:=FALSE;
END_IF
//******污水泵和污水泵球阀控制******
R_HMI_wastewater_pump(CLK:=HMI_wastewater_pump);
R_T_DI_auxiliary1_warte_H(CLK:=T_DI_auxiliary1_warte_H.Q);
R_T_DI_auxiliary2_warte_H(CLK:=T_DI_auxiliary2_warte_H.Q);
IF (R_HMI_wastewater_pump.Q OR R_auto_wastewater_pump.Q) AND (NOT ASweeproad_HMI) AND (NOT LSweeproad_HMI) AND (NOT RSweeproad_HMI)AND (NOT DO_wastewater_pump_open100) THEN
	DO_wastewater_pump_open1:=TRUE;
ELSIF (R_HMI_wastewater_pump.Q OR R_T_DI_auxiliary1_warte_H.Q OR R_T_DI_auxiliary2_warte_H.Q OR F_Motor_Work.Q OR R_T_DO_wastewater_pump_open1.Q) AND DO_wastewater_pump_open100 THEN
	DO_wastewater_pump_open1:=FALSE;
END_IF
DO_wastewater_pump_open100:=DO_wastewater_pump_open1;
T_DO_wastewater_pump_open1(IN:=DO_wastewater_pump_open1,PT:=T#600S);//10分钟延时
R_T_DO_wastewater_pump_open1(CLK:=T_DO_wastewater_pump_open1.Q);//污水泵打开10分钟后上升沿
R_auto_wastewater_pump(CLK:=T_DI_wastewater_full.Q AND NOT Wastewater_full_Fault AND motor_work AND (NOT T_DO_wastewater_pump_open1.Q));//自动排污上升沿
//污水泵球阀打开标志
T_DO_wastewater_valve_open(IN:=DO_wastewater_pump_open1,PT:=T#3S);
//高压冲洗启停控制
R_HMI_Hpre_wash(CLK:=HMI_Hpre_wash);//高压冲洗上升沿
R_Func_test_HMI(CLK:=Func_test_HMI);//功能测试上升沿
IF R_HMI_Hpre_wash.Q AND NOT Func_test_HMI AND motor_work AND Hpre_waterpump_open_pre AND NOT DO_Hpressure_water100 THEN
	DO_Hpressure_water1:=TRUE;
ELSIF (R_HMI_Hpre_wash.Q OR R_Func_test_HMI.Q OR F_Motor_Work.Q OR (F_Hpre_waterpump_open_pre.Q AND (NOT Func_test_HMI)))AND DO_Hpressure_water100 THEN
	DO_Hpressure_water1:=FALSE;
END_IF
DO_Hpressure_water100:=DO_Hpressure_water1;
//自洁启停控制
R_HMI_selfclean(CLK:=HMI_selfclean);//自洁上升沿
IF R_HMI_selfclean.Q AND NOT Func_test_HMI AND motor_work AND Hpre_waterpump_open_pre AND NOT DO_selfclean_water100 THEN
	DO_selfclean_water1:=TRUE;
ELSIF (R_HMI_selfclean.Q OR R_Func_test_HMI.Q OR F_Motor_Work.Q OR (F_Hpre_waterpump_open_pre.Q AND (NOT Func_test_HMI)))AND DO_selfclean_water100 THEN
	DO_selfclean_water1:=FALSE;
END_IF
DO_selfclean_water100:=DO_selfclean_water1;
//*****高压水泵起停控制*****
//高压水泵打开条件标志位M79
Hpre_waterpump_open_pre:=Totvalve_open_sign AND Hpre_valve_sign AND (NOT T_water_overflow_noClose.Q) AND (NOT T_DI_cleanwater_LOW.Q) AND (NOT T_Pumpspeed_HH.Q) AND Motor_work AND (NOT T_DI_air_press_low.Q);
F_Hpre_waterpump_open_pre(CLK:=Hpre_waterpump_open_pre);//高压水泵打开条件下降沿
//高压水泵打开中间变量M78
Hpre_waterpump_open_Mid:=T_DO_Suction_water.Q OR T_DO_Lrod_water.Q OR T_DO_Rrod_water.Q OR DO_Hpressure_water1 OR DO_selfclean_water1 OR Hpre_waterpump_open_pre1;
//高压水泵提前启动寄存器
Hpre_waterpump_open_pre1:=AwashSweep_HMI OR LwashSweep_HMI OR RwashSweep_HMI OR Aclean_HMI OR Rclean_HMI OR Lclean_HMI;
//高压水泵未啮合提示
DO_Hpre_pump_noWork:=Hpre_waterpump_open_Mid AND NOT Hpre_waterpump_open_pre;
//高压水路球阀未打开
DI_Totvalve_noOpen:=Hpre_waterpump_open_Mid AND NOT DI_Totvalve_Open;
//高压吹净球阀未打开提示
DI_Hpre_valve_noOpen:=Hpre_waterpump_open_Mid AND NOT DI_Hpre_valve_Open;

//高压冲洗速度给定
R_DO_Hpressure_water1(CLK:=DO_Hpressure_water1);// 高压冲洗标志位上升沿
IF R_DO_Hpressure_water1.Q AND Motor_work THEN
	SETspeed_PID:=S_Idle_Speed;(* 把怠速给设定速度 *)
END_IF
//自洁速度给定
R_DO_selfclean_water1(CLK:=DO_selfclean_water1);// 自洁标志位上升沿
IF R_DO_selfclean_water1.Q AND Motor_work THEN
	SETspeed_PID:=1200;(* 把1200给设定速度 *)
END_IF
//自洁和高压冲洗关闭时速度给定
F_DO_Hpressure_water1(CLK:=DO_Hpressure_water1);// 高压冲洗标志位下降沿
F_DO_selfclean_water1(CLK:=DO_selfclean_water1);// 自洁标志位下降沿
IF ((F_DO_Hpressure_water1.Q AND NOT DO_selfclean_water1) OR (F_DO_selfclean_water1.Q AND NOT DO_Hpressure_water1))AND NOT sys_work AND motor_work THEN
	SETspeed_PID:=S_Idle_Speed;(* 把怠速给设定速度 *)
END_IF

//系统工作时，给定标准转速

F_Intelligent_HMI(CLK:=Intelligent_HMI);//智能标志下降沿
IF (R_sys_work.Q AND NOT Intelligent_HMI) OR (F_Intelligent_HMI.Q AND sys_work) THEN
	SETspeed_PID:=S_Standard_Speed;(* 把副发标准速度给PID给定速度 *)
END_IF
R_sys_work(CLK:=sys_work);//系统工作上升沿
//存储原始速度，再怠速调整
R_Hpre_waterpump_open_Mid(CLK:=Hpre_waterpump_open_Mid);
IF R_Hpre_waterpump_open_Mid.Q AND Hpre_waterpump_open_Mid AND Hpre_waterpump_open_pre AND NOT Hpre_waterpump_open_Mid2 THEN
	Hpre_waterpump_open_Mid1:=TRUE;
ELSIF (NOT Hpre_waterpump_open_Mid) OR (NOT Hpre_waterpump_open_pre) OR Hpre_waterpump_open_Mid2  THEN
	Hpre_waterpump_open_Mid1:=FALSE;
END_IF
R_Hpre_waterpump_open_Mid1(CLK:=Hpre_waterpump_open_Mid1);
IF R_Hpre_waterpump_open_Mid1.Q THEN
	SETspeed_1:=SETspeed_PID;(* 把设定速度给暂存值 *)
END_IF

IF R_Hpre_waterpump_open_Mid1.Q AND motor_work THEN
	SETspeed_PID:=S_Idle_Speed;(* 把怠速给设定速度 *)
END_IF
IF Hpre_waterpump_open_Mid1 THEN
	SETspeed_2:=Motor_real_speed_HMI-S_Idle_Speed;(* 把怠速给设定速度 *)
END_IF
Speed_Dif:=(SETspeed_2 < 30);//实际值与给定值的偏差
T_Hpre_waterpump_open_Mid1(IN:=Hpre_waterpump_open_Mid1,PT:=T#10S);
//高压水泵啮合过程
R_Speed_Dif(CLK:=Speed_Dif);
R_T_Hpre_waterpump_open_Mid1(CLK:=T_Hpre_waterpump_open_Mid1.Q);
IF (R_Speed_Dif.Q OR R_T_Hpre_waterpump_open_Mid1.Q)AND Hpre_waterpump_open_Mid AND Hpre_waterpump_open_pre AND NOT T_Hpre_waterpump_open_Mid2.Q THEN
	Hpre_waterpump_open_Mid2:=TRUE;
ELSIF NOT Hpre_waterpump_open_Mid OR NOT Hpre_waterpump_open_pre OR T_Hpre_waterpump_open_Mid2.Q THEN
	Hpre_waterpump_open_Mid2:=FALSE;
END_IF
T_Hpre_waterpump_open_Mid2(IN:=Hpre_waterpump_open_Mid2,PT:=T#3S);
//高压水泵打开
F_Hpre_waterpump_open_Mid(CLK:=Hpre_waterpump_open_Mid);//m78下降沿
IF Hpre_waterpump_open_Mid2 THEN
	DO_Hpre_pump1:=TRUE;
ELSIF F_Hpre_waterpump_open_Mid.Q OR F_Hpre_waterpump_open_pre.Q THEN
	DO_Hpre_pump1:=FALSE;
END_IF
R_T_Hpre_waterpump_open_Mid2(CLK:=T_Hpre_waterpump_open_Mid2.Q);
IF R_T_Hpre_waterpump_open_Mid2.Q AND motor_work THEN
	SETspeed_PID:=SETspeed_1;(* 把暂存值给设定速度 *)
END_IF

//垃圾箱门开关控制
DO_Door_Close1:=HMI_Door_Close AND NOT HMI_Door_Open;
DO_Door_Open1:=HMI_Door_Open AND NOT HMI_Door_Close;
//垃圾箱升级控制
DO_Box_Up1:=NOT DI_box_door_close AND HMI_Box_Up;
DO_Box_Up_arm:=DI_box_door_close AND HMI_Box_Up;
DO_Box_Down1:=NOT DI_Rod_noDown AND HMI_Box_Down;
DO_Box_Down_arm:=DI_Rod_noDown AND HMI_Box_Down;

//电机启停控制
IF HMI_start_motor AND NOT HMI_stop_motor THEN
	motor_start:=TRUE;
ELSIF HMI_stop_motor AND NOT HMI_start_motor THEN
	motor_start:=FALSE;	//用于电机停止给定速度
END_IF
//底盘未上高压提醒
High_voltage_noReady:=HMI_start_motor AND NOT High_voltage_Ready;
//电机启动条件
T_HMI_start_motor(IN:=HMI_start_motor AND High_voltage_Ready,PT:=T#25S);
motor_start_Mid:=HMI_start_motor AND High_voltage_Ready AND NOT motor_work AND NOT HMI_stop_motor AND NOT T_HMI_start_motor.Q;
//启动触发，5S后启动马达
T_HMI_start_motor1(IN:=motor_start_Mid AND NOT DI_backup_power_open,PT:=T#5S);//启动触发5S后马达得电
R_T_HMI_start_motor1(CLK:=T_HMI_start_motor1.Q);
R_Sweep_stop_HMI(CLK:=Sweep_stop_HMI);//
IF R_T_HMI_start_motor1.Q OR (R_Sweep_stop_HMI.Q AND motor_work) THEN
	SETspeed_PID:=S_Idle_Speed;(* 把怠速给设定速度 *)
END_IF
//启动按钮后3.5内还没转速，则停机
IF R_T_HMI_start_motor1.Q THEN
	HMI_start_motor_overT :=TRUE;
ELSIF T_HMI_start_motor_overT.Q THEN
	HMI_start_motor_overT :=FALSE;
END_IF
T_HMI_start_motor_overT(IN:=HMI_start_motor_overT,PT:=T#8S);
IF T_HMI_start_motor_overT.Q AND NOT motor_work THEN
	SETspeed_PID:=0;(* 把零给设定速度 *)
	motor_start:=FALSE;	//用于电机停止给定速度
END_IF
//电机停止控制
R_backup_power_stopmotor(CLK:=DI_backup_power_open AND motor_work);//备用动力开关触发停机
R_T_Motor_CAN_fault(CLK:=T_Motor_CAN_fault.Q);
IF R_backup_power_stopmotor.Q OR HMI_stop_motor OR (NOT High_voltage_Ready) OR T_Chassis_SOC_LOW.Q OR T_motor_fault.Q OR R_T_Motor_CAN_fault.Q OR T_HMI_MOTOR_runstop_M.Q THEN
   SETspeed_PID:=0;(* 把零给设定速度 *)
   	
END_IF
R_motor_stop(CLK:=motor_stop);
IF R_motor_stop.Q THEN
   motor_stop:=FALSE;
   Intelligent_HMI:=FALSE;(* 智能 *)
   Cleanly_HMI:=FALSE;(* 清洁 *)
   Normal_HMI:=FALSE;(* 一般 *)
   Dirty_HMI :=FALSE;(* 污染 *) 
END_IF





T_motor_fault(IN:=(SETspeed_PID>250) AND (Motor_real_speed_HMI<50),PT:=T#10S);//电机故障停机的判断

//电机水冷泵控制，风扇控制
IF motor_work AND (NOT T_DO_watercooler_pump_open1.Q) THEN
	DO_watercooler_pump_open1:=TRUE;
	DO_cooler_fan_open1:=TRUE;
ELSIF T_DO_watercooler_pump_open1.Q THEN
	DO_watercooler_pump_open1:=FALSE;
	DO_cooler_fan_open1:=FALSE;	
END_IF
T_DO_watercooler_pump_open1(IN:=DO_watercooler_pump_open1 AND (NOT motor_work),PT:=T#6S);



//电机标准强力速度切换
R_HMI_Standard_speed(CLK:=HMI_Standard_speed);//标准工作速度上升沿
R_HMI_Strong_speed(CLK:=HMI_Strong_speed);//强力工作速度上升沿
IF R_HMI_Standard_speed.Q AND NOT HMI_Strong_speed AND motor_work AND NOT Intelligent_HMI THEN
	SETspeed_PID:=S_Standard_Speed;(* 把副发标准速度给PID给定速度 *)
END_IF
IF R_HMI_Strong_speed.Q AND NOT HMI_Standard_speed AND motor_work AND NOT Intelligent_HMI THEN
	SETspeed_PID:=S_Strong_Speed;(* 把副发强力速度给PID给定速度 *)
END_IF
IF R_HMI_Strong_speed.Q AND NOT HMI_Standard_speed AND motor_work AND NOT Intelligent_HMI AND (Hpre_waterpump_open_Mid1 OR Hpre_waterpump_open_Mid2) THEN
	SETspeed_1:=S_Strong_Speed;(* 把副发强力速度给PID给定速度 *)
END_IF
//标准和强力标志
Standard_speed_HMI:=(SETspeed_PID=S_Standard_Speed) AND NOT Intelligent_HMI;
Strong_speed_HMI:=(SETspeed_PID=S_Strong_Speed) AND NOT Intelligent_HMI;

//电机速度加减控制
R_HMI_Inc_Speed(CLK:=HMI_Inc_Speed);//电机加速上升沿
R_HMI_Dec_Speed(CLK:=HMI_Dec_Speed);//电机减速上升沿
//速度加
IF NOT Intelligent_HMI AND motor_work AND R_HMI_Inc_Speed.Q THEN
	SETspeed_PID:=SETspeed_PID+S_IncDec_Speed;
END_IF
IF NOT Intelligent_HMI AND motor_work AND R_HMI_Inc_Speed.Q AND (SETspeed_PID>=S_MAX_Speed) THEN
	SETspeed_PID:=S_MAX_Speed;
END_IF
//速度减
IF NOT Intelligent_HMI AND motor_work AND R_HMI_Dec_Speed.Q THEN
	SETspeed_PID:=SETspeed_PID-S_IncDec_Speed;
END_IF
IF NOT Intelligent_HMI AND motor_work AND R_HMI_Dec_Speed.Q AND (SETspeed_PID<=S_min_speed) THEN
	SETspeed_PID:=S_min_speed;
END_IF

//扫盘速度控制
R_HMI_Sweep_Hspd(CLK:=HMI_Sweep_Hspd);//高速上升沿
R_HMI_Sweep_Mspd(CLK:=HMI_Sweep_Mspd);//中速上升沿
R_HMI_Sweep_Lspd(CLK:=HMI_Sweep_Lspd);//低速上升沿
IF R_HMI_Sweep_Hspd.Q AND NOT HMI_Sweep_Mspd AND NOT HMI_Sweep_Lspd THEN
    Sweep_HSpeed_HMI:=TRUE;(* 扫盘高速 *)
    Sweep_MSpeed_HMI:=FALSE;(* 扫盘中速 *)
    Sweep_LSpeed_HMI:=FALSE;(* 扫盘低速 *)	
END_IF
IF R_HMI_Sweep_Mspd.Q AND NOT HMI_Sweep_Hspd AND NOT HMI_Sweep_Lspd THEN
    Sweep_HSpeed_HMI:=FALSE;(* 扫盘高速 *)
    Sweep_MSpeed_HMI:=TRUE;(* 扫盘中速 *)
    Sweep_LSpeed_HMI:=FALSE;(* 扫盘低速 *)	
END_IF
IF R_HMI_Sweep_Lspd.Q AND NOT HMI_Sweep_Hspd AND NOT HMI_Sweep_Mspd THEN
    Sweep_HSpeed_HMI:=FALSE;(* 扫盘高速 *)
    Sweep_MSpeed_HMI:=FALSE;(* 扫盘中速 *)
    Sweep_LSpeed_HMI:=TRUE;(* 扫盘低速 *)	
END_IF

//点喷控制
Pointshoot_up_HMI:=HMI_pointshoot_up AND NOT HMI_pointshoot_down;
Pointshoot_down_HMI:=HMI_pointshoot_down AND NOT HMI_pointshoot_up;
Pointshoot_left_HMI:=HMI_pointshoot_left AND NOT HMI_pointshoot_right;
Pointshoot_right_HMI:=HMI_pointshoot_right AND NOT HMI_pointshoot_left;



//*************以下为智能控制程序段*************
//底盘车速级别判断
T_Chassis_stop(IN:=Chassis_speed<1,PT:=T#1S);//车停
T_Chassis_Lspeed(IN:=0<Chassis_speed AND Chassis_speed<=8,PT:=T#1S);//车辆低速
T_Chassis_M_Lspeed(IN:=8<Chassis_speed AND Chassis_speed<=12,PT:=T#1S);//车辆中低速
T_Chassis_M_Hspeed(IN:=12<Chassis_speed AND Chassis_speed<=16,PT:=T#1S);//车辆中高速
T_Chassis_Hspeed(IN:=16<Chassis_speed,PT:=T#1S);//车辆高速
//智能输入操作
R_HMI_intelligent(CLK:=HMI_intelligent);//智能上升沿
R_HMI_cleanly(CLK:=HMI_cleanly);// 清洁上升沿
R_HMI_normal(CLK:=HMI_normal);// 一般上升沿
R_HMI_dirty(CLK:=HMI_dirty);// 污染上升沿
F_sys_work(CLK:=sys_work);//系统工作下降沿
IF R_HMI_intelligent.Q AND NOT Intelligent_HMI100 THEN
    Intelligent_HMI:=TRUE;	
ELSIF (R_HMI_intelligent.Q AND Intelligent_HMI100) OR F_Motor_Work.Q THEN
    Intelligent_HMI:=FALSE;(* 智能 *)
    Cleanly_HMI:=FALSE;(* 清洁 *)
    Normal_HMI:=FALSE;(* 一般 *)
    Dirty_HMI :=FALSE;(* 污染 *)  	
END_IF
Intelligent_HMI100:=Intelligent_HMI;	
//清洁
IF R_HMI_cleanly.Q AND Intelligent_HMI THEN
    Cleanly_HMI:=TRUE;(* 清洁 *)
    Normal_HMI:=FALSE;(* 一般 *)
    Dirty_HMI :=FALSE;(* 污染 *)  	
END_IF
//一般
R_Intelligent_HMI(CLK:=Intelligent_HMI);
IF (R_HMI_normal.Q AND Intelligent_HMI) OR R_Intelligent_HMI.Q THEN
    Cleanly_HMI:=FALSE;(* 清洁 *)
    Normal_HMI:=TRUE;(* 一般 *)
    Dirty_HMI :=FALSE;(* 污染 *)  	
END_IF
//污染
IF R_HMI_dirty.Q AND Intelligent_HMI THEN
    Cleanly_HMI:=FALSE;(* 清洁 *)
    Normal_HMI:=FALSE;(* 一般 *)
    Dirty_HMI :=TRUE;(* 污染 *) 	
END_IF
//不同状况下的转速设定值
//*******低速或车停时
//清洁路面
IF sys_work AND Cleanly_HMI AND (T_Chassis_stop.Q OR T_Chassis_Lspeed.Q) THEN
	SETspeed_PID:=S_clean_low_speed;(*清洁低速速度*)
END_IF
//一般路面
IF sys_work AND Normal_HMI AND (T_Chassis_stop.Q OR T_Chassis_Lspeed.Q) THEN
	SETspeed_PID:=S_normal_low_speed;(*一般低速速度*)
END_IF
//污染路面
IF sys_work AND Dirty_HMI AND (T_Chassis_stop.Q OR T_Chassis_Lspeed.Q) THEN
	SETspeed_PID:=S_dirty_low_speed;(*污染低速速度*)
END_IF

//*******中低速时
//清洁路面
IF sys_work AND Cleanly_HMI AND T_Chassis_M_Lspeed.Q THEN
	SETspeed_PID:=S_clean_midlow_speed;(*清洁中低速速度*)
END_IF
//一般路面
IF sys_work AND Normal_HMI AND T_Chassis_M_Lspeed.Q THEN
	SETspeed_PID:=S_normal_midlow_speed;(*一般中低速速度*)
END_IF
//污染路面
IF sys_work AND Dirty_HMI AND T_Chassis_M_Lspeed.Q THEN
	SETspeed_PID:=S_dirty_midlow_speed;(*污染中低速速度*)
END_IF

//*******中高速时
//清洁路面
IF sys_work AND Cleanly_HMI AND T_Chassis_M_Hspeed.Q THEN
	SETspeed_PID:=S_clean_midhigh_speed;(*清洁中高速速度*)
END_IF
//一般路面
IF sys_work AND Normal_HMI AND T_Chassis_M_Hspeed.Q THEN
	SETspeed_PID:=S_normal_midhigh_speed;(*一般中高速速度*)
END_IF
//污染路面
IF sys_work AND Dirty_HMI AND T_Chassis_M_Hspeed.Q THEN
	SETspeed_PID:=S_dirty_midhigh_speed;(*污染中高速速度*)
END_IF

//********高速时
//清洁路面
IF sys_work AND Cleanly_HMI AND T_Chassis_Hspeed.Q THEN
	SETspeed_PID:=S_clean_high_speed;(*清洁高速速度*)
END_IF
//一般路面
IF sys_work AND Normal_HMI AND T_Chassis_Hspeed.Q THEN
	SETspeed_PID:=S_normal_high_speed;(*一般高速速度*)
END_IF
//污染路面
IF sys_work AND Dirty_HMI AND T_Chassis_Hspeed.Q THEN
	SETspeed_PID:=S_dirty_high_speed;(*污染高速速度*)
END_IF

//**********检修盒控制***********
//扫盘升降
JX_Sweep_up:=DI_Sweep_Up AND NOT Func_test_HMI AND NOT Sys_work AND NOT DI_Sweep_Down;
JX_Sweep_Down:=DI_Sweep_Down AND NOT Func_test_HMI AND NOT Sys_work AND NOT DI_Sweep_Up;
//扫盘摆出
IF DI_sweep_out AND NOT Func_test_HMI AND NOT Sys_work AND NOT DI_sweep_return THEN
	JX_Sweep_out:=TRUE;
END_IF
IF DI_sweep_return AND NOT Func_test_HMI AND NOT Sys_work AND NOT DI_sweep_out THEN
	JX_Sweep_out:=FALSE;	
END_IF
(*JX_Sweep_out:=DI_sweep_out AND NOT Func_test_HMI AND NOT Sys_work AND NOT DI_sweep_return;
JX_Sweep_return:=DI_sweep_return AND NOT Func_test_HMI AND NOT Sys_work AND NOT DI_sweep_out;*)
//备用动力
T_DI_oil_release_valve(IN:=NOT DI_oil_release_valve,PT:=T#3.5S);//车停
IF DI_oil_release_valve AND NOT T_DI_oil_release_valve.Q AND DI_backup_power_open THEN
	JX_backup_power_open:=TRUE;
ELSIF T_DI_oil_release_valve.Q OR NOT DI_backup_power_open THEN
	JX_backup_power_open:=FALSE;
END_IF

//电机停止按钮或者没有高压时，禁止电机启动
k:=FALSE;
IF NOT motor_start OR NOT High_voltage_Ready THEN
	SETspeed_PID:=0;
	k:=TRUE;
END_IF

//更换扫刷
R_HMI_replace_Sweep(CLK:=HMI_replace_Sweep);
IF R_HMI_replace_Sweep.Q AND NOT motor_work AND NOT replace_Sweep_HMI1 THEN
	replace_Sweep_HMI:=TRUE;
	ELSIF (R_HMI_replace_Sweep.Q AND replace_Sweep_HMI1) OR HMI_start_motor THEN
	replace_Sweep_HMI:=FALSE;	
END_IF
replace_Sweep_HMI1:=replace_Sweep_HMI;	

//冬季排水启停控制
R_HMI_drain_start(CLK:=HMI_drain_start);//冬季排水上升沿
IF R_HMI_drain_start.Q AND NOT motor_work AND NOT Drain_start_HMI100 THEN
	Drain_start_HMI:=TRUE;
	ELSIF (R_HMI_drain_start.Q AND Drain_start_HMI100) OR HMI_start_motor THEN
	Drain_start_HMI:=FALSE;
END_IF
Drain_start_HMI100:=Drain_start_HMI;
//冬季排水手动
R_HMI_drain_manual(CLK:=HMI_drain_manual);//手动排水上升沿
IF R_HMI_drain_manual.Q AND NOT motor_work AND Drain_start_HMI AND NOT Drain_manual_HMI100 THEN
	Drain_manual_HMI:=TRUE;
	ELSIF (R_HMI_drain_manual.Q AND Drain_manual_HMI100) OR NOT Drain_start_HMI OR R_HMI_drain_auto.Q OR HMI_start_motor THEN
	Drain_manual_HMI:=FALSE;	
END_IF
Drain_manual_HMI100:=Drain_manual_HMI;
//手动排水
Lrod_drain_HMI_manu:=Drain_manual_HMI AND Drain_start_HMI AND HMI_Lrod_drain;//左喷杆排水手动中间变量
Rrod_drain_HMI_manu:=Drain_manual_HMI AND Drain_start_HMI AND HMI_Rrod_drain;//右喷杆排水手动中间变量
Suction_drain_HMI_manu:=Drain_manual_HMI AND Drain_start_HMI AND HMI_Suction_drain;//吸嘴排水手动中间变量
Hpressure_drain_HMI_manu:=Drain_manual_HMI AND Drain_start_HMI AND HMI_Hpressure_drain;//高辅排水手动中间变量
Selfclean_drain_HMI_manu:=Drain_manual_HMI AND Drain_start_HMI AND HMI_selfclean_drain;//自洁排水手动中间变量

//冬季排水自动
R_HMI_drain_auto(CLK:=HMI_drain_auto);//冬季排水上升沿
IF R_HMI_drain_auto.Q AND NOT motor_work AND Drain_start_HMI AND NOT Drain_auto_HMI100 THEN
	Drain_auto_HMI:=TRUE;
	ELSIF (R_HMI_drain_auto.Q AND Drain_auto_HMI100) OR NOT Drain_start_HMI OR R_HMI_drain_manual.Q OR HMI_start_motor OR T_Selfclean_drain_HMI_auto.Q THEN
	Drain_auto_HMI:=FALSE;	
END_IF
Drain_auto_HMI100:=Drain_auto_HMI;
T_Lrod_drain_HMI_auto(IN:=Drain_start_HMI AND Drain_auto_HMI,PT:=T#4S);//排水时间
T_Rrod_drain_HMI_auto(IN:=T_Lrod_drain_HMI_auto.Q,PT:=T#4S);//排水时间
T_Suction_drain_HMI_auto(IN:=T_Rrod_drain_HMI_auto.Q,PT:=T#4S);//排水时间
T_Hpressure_drain_HMI_auto(IN:=T_Suction_drain_HMI_auto.Q,PT:=T#4S);//排水时间
T_Selfclean_drain_HMI_auto(IN:=T_Hpressure_drain_HMI_auto.Q,PT:=T#4S);//排水时间
//自动排水
Lrod_drain_HMI_auto:=NOT T_Lrod_drain_HMI_auto.Q AND Drain_start_HMI AND Drain_auto_HMI;//左喷杆自动排水
Rrod_drain_HMI_auto:=T_Lrod_drain_HMI_auto.Q AND NOT T_Rrod_drain_HMI_auto.Q;//右喷杆自动排水
Suction_drain_HMI_auto:=T_Rrod_drain_HMI_auto.Q AND NOT T_Suction_drain_HMI_auto.Q;//吸嘴自动排水
Hpressure_drain_HMI_auto:=T_Suction_drain_HMI_auto.Q AND NOT T_Hpressure_drain_HMI_auto.Q;//高辅自动排水
Selfclean_drain_HMI_auto:=T_Hpressure_drain_HMI_auto.Q AND NOT T_Selfclean_drain_HMI_auto.Q;//自洁自动排水
//排水标志位
Lrod_drain_HMI:=Lrod_drain_HMI_manu OR Lrod_drain_HMI_auto;//左喷杆排水标志位
Rrod_drain_HMI:=Rrod_drain_HMI_manu OR Rrod_drain_HMI_auto;
Suction_drain_HMI:=Suction_drain_HMI_manu OR Suction_drain_HMI_auto;
Hpressure_drain_HMI:=Hpressure_drain_HMI_manu OR Hpressure_drain_HMI_auto;
Selfclean_drain_HMI:=Selfclean_drain_HMI_manu OR Selfclean_drain_HMI_auto;

//与屏通信超时，复位屏输入按钮 
//与屏CAN通讯失败后，停止动作和电机
T_HMI_MOTOR_runstop_M(IN:=HMI_MOTOR_runstop_M,PT:=T#8S);(* 超时触发停机 *)
IF T_HMI_MOTOR_runstop_M.Q THEN
   SETspeed_PID:=0;(* 副发运行停止 *)
   motor_start:=FALSE;
   HMI_MOTOR_runstop_M:=FALSE;(* 屏通信失败停扫 *)
END_IF

IF T_Screen_CAN_fault.Q THEN
   AwashSweep_HMI:=FALSE;(* 全洗扫 *)
   LwashSweep_HMI:=FALSE;(* 左洗扫 *)
   RwashSweep_HMI:=FALSE;(* 右洗扫 *)
   ASweeproad_HMI:=FALSE;(* 全扫路 *)
   LSweeproad_HMI:=FALSE;(* 左扫路 *)
   RSweeproad_HMI:=FALSE;(* 右扫路 *)
   Aclean_HMI:=FALSE;(* 全清洗 *)
   Lclean_HMI:=FALSE;(* 左清洗 *)
   Rclean_HMI:=FALSE;(* 右清洗 *)
   Sweep_stop_HMI:=FALSE;(* 停扫 *)
   Intelligent_HMI:=FALSE;(* 智能 *)
   Cleanly_HMI:=FALSE;(* 清洁 *)
   Normal_HMI:=FALSE;(* 一般 *)
   Dirty_HMI :=FALSE;(* 污染 *) 
   DO_Rsweep_out1:=FALSE; 
   DO_Lsweep_down1:=FALSE;
   DO_Lsweep_up1:=FALSE;
   DO_Rsweep_down1:=FALSE;
   DO_Rsweep_up1:=FALSE;
   DO_Lsweep_out1:=FALSE;
   DO_Rsweep_out1:=FALSE;
   DO_Lrod_out1:=FALSE;
   DO_Rrod_out1:=FALSE;
   DO_Hpressure_water1:=FALSE;
   DO_selfclean_water1:=FALSE;
   DO_Hpre_pump1:=FALSE;
   DO_fog_Spump1:=FALSE;
   DO_wastewater_pump_open1:=FALSE;
   LSweep:=FALSE;
   RSweep:=FALSE;
   ASweep:=FALSE;
   HMI_MOTOR_runstop_M:=TRUE;(* 屏通信失败停扫 *)
END_IF




//输出控制
DO_Lsweep_down:=LSweep_Down_Test OR DO_Lsweep_down1 OR JX_Sweep_Down;//左扫盘下降
DO_Lsweep_up:=LSweep_Up_Test OR DO_Lsweep_up1 OR JX_Sweep_up;//左扫盘上升
DO_Rsweep_down:=RSweep_Down_Test OR DO_Rsweep_down1 OR JX_Sweep_Down;//右扫盘下降
DO_Rsweep_up:=RSweep_Up_Test OR DO_Rsweep_up1 OR JX_Sweep_up;//左扫盘上升
DO_Lsweep_out:=LSweep_out_Test OR DO_Lsweep_out1 OR JX_Sweep_out;//左扫盘摆出
DO_Rsweep_out:=RSweep_out_Test OR DO_Rsweep_out1 OR JX_Sweep_out;//右扫盘摆出
DO_Lrod_out:=Lrod_OUT_Test OR DO_Lrod_out1;//左喷杆摆出
DO_Rrod_out:=Rrod_OUT_Test OR DO_Rrod_out1;//右喷杆摆出
DO_water_overflow:=DO_Lrod_water OR DO_Rrod_water OR DO_Suction_water OR DO_Hpressure_water OR DO_selfclean_water;//水泵卸荷阀
DO_Lrod_water:=Lrod_water_Test OR T_DO_Lrod_water.Q OR Lrod_drain_HMI;//左喷杆球阀打开
DO_Rrod_water:=Rrod_water_Test OR T_DO_Rrod_water.Q OR Rrod_drain_HMI;//右喷杆球阀打开
DO_Suction_water:=Suction_water_Test OR T_DO_Suction_water.Q OR Suction_drain_HMI;//吸嘴喷杆球阀打开
DO_Hpressure_water:=Hpre_wash_Test OR DO_Hpressure_water1 OR Hpressure_drain_HMI;//高压辅助球阀打开
DO_selfclean_water:=selfclean_water_Test OR DO_selfclean_water1 OR Selfclean_drain_HMI;//自洁球阀打开
DO_Hpre_pump:=Hpress_pump_gearin_Test OR DO_Hpre_pump1;//高压水泵离合器啮合
DO_fog_Spump:=(Fog_pump_Test OR DO_fog_Spump1) AND DI_fog_pump_press_ok;//低压隔膜泵启停
//DO_Motor_en  电机使能
DO_watercooler_pump:=cooler_motor_Test OR DO_watercooler_pump_open1;//水冷泵电机控制
DO_cooler_fan:=cooler_fan_Test OR DO_cooler_fan_open1;//散热风扇控制
DO_backup_power:=Backup_power_Test OR JX_backup_power_open;//备用动力控制
DO_wastewater_valve:=Wastewater_valve_Test OR T_DO_wastewater_valve_open.Q;//污水泵球阀打开
DO_wastewater_pump:=Wastewater_pump_Test OR DO_wastewater_pump_open1;//污水泵打开
DO_oil_release_valve:=DO_RSweep OR DO_LASweep OR DO_RASweep OR DO_Box_Down OR DO_Box_Up OR DO_Suction_Down OR DO_Suction_Up OR DO_Door_Open OR DO_Door_Close;//油路卸荷阀
DO_Sweep_Mspeed:=Sweep_Mspeed_Test OR ((LSweep OR RSweep OR ASweep)AND Sweep_MSpeed_HMI);//扫盘中速
DO_Sweep_Lspeed:=Sweep_Lspeed_Test OR ((LSweep OR RSweep OR ASweep)AND Sweep_LSpeed_HMI);//扫盘低速
DO_RSweep:=RSweep_Test OR RSweep;//右扫旋转
DO_LASweep:=LSweep_Test OR LSweep OR ASweep_Test OR ASweep;//左全扫旋转
DO_RASweep:=RSweep_Test OR RSweep OR ASweep_Test OR ASweep OR replace_Sweep_HMI;//右全扫旋转
DO_Box_Down:=Box_Down_Test OR DO_Box_Down1;//箱体降
DO_Box_Up:=Box_Up_Test OR DO_Box_Up1;//箱体升
DO_Suction_Down:=Suction_Down_Test OR DO_Suction_Down1;//吸盘降
DO_Suction_Up:=Suction_Up_Test OR DO_Suction_Up1;//吸盘升
DO_Door_Open:=Boxdoor_open_Test OR DO_Door_Open1;//箱门开
DO_Door_Close:=Boxdoor_close_Test OR DO_Door_Close1;//箱门关
DO_pointshoot_up := Pointshoot_up_Test OR Pointshoot_up_HMI;//点喷上
DO_pointshoot_down := Pointshoot_down_Test OR Pointshoot_down_HMI;//点喷下
DO_pointshoot_left := Pointshoot_left_Test OR Pointshoot_left_HMI;//点喷左
DO_pointshoot_right := Pointshoot_right_Test OR Pointshoot_right_HMI;//点喷右

END_PROGRAM

// Changsha_Xiangji_ARM_Cortex_A9_xilinx_zynq7000_linux/Application/parameters/fn_write_para_file
FUNCTION fn_write_para_file : BOOL
VAR_INPUT
	para:ST_PARA;	
END_VAR
VAR
	bak_file_prefix:STRING :=ANY_TO_STRING("parameters_bak_");
	bak_file:STRING := ANY_TO_STRING("");	
	hFile: RTS_IEC_HANDLE;
	udiDeleteError: RTS_IEC_RESULT;
	udiOpenError: RTS_IEC_RESULT;
	udiWriteError: RTS_IEC_RESULT;
	filesize: __XWORD;
	i :UINT;
	iTemp: UDINT;
	udiPos: UDINT;
	str: STRING(256);
	str_size: __XWORD;
	udiByteWrite: __XWORD;
	check_sum:REAL := 0;
	gRandomNum :LWORD := 1;   //系统随机数,每个周期乘以内部传感器的实时值；
END_VAR

fn_write_para_file := FALSE;
gRandomNum := (gRandomNum+1359+ %ID57)*%ID49;

IF para.len = 0 THEN
	RETURN;
END_IF

//检测文件是否存在，如果存在自动备份
hFile := sysfileopen(szFile := gvl.para_file, am := sysfile.AM_READ, pResult:= ADR(udiOpenError));
IF hFile <> RTS_INVALID_HANDLE	THEN  //文件存在
	sysfile.SysFileClose(hFile);  
	bak_file := concat(str1 := bak_file_prefix, str2:= ANY_TO_STRING(gRandomNum));
	filesize := para.len*16;
	sysfile.SysFileCopy(szDestFileName := bak_file, szSourceFileName := gvl.para_file, pulCopied := ADR(filesize));
	sysfile.SysFileDelete(szFileName := gvl.para_file);
END_IF

hFile := sysfileopen(szFile := gvl.para_file, am := sysfile.AM_WRITE, pResult := ADR(udiOpenError));
IF hFile <> RTS_INVALID_HANDLE THEN //创建文件成功
	udiPos := SysFileSetPos(hFile:=hFile, ulOffset:=0);	
	
	check_sum := 0;
	str:= ANY_TO_STRING("");
	FOR i := 0 TO para.len DO
		str := concat(str, ANY_TO_STRING(para.para_val[i]));
		str := concat(str, ANY_TO_STRING(","));
		check_sum := check_sum + para.para_val[i];		
	END_FOR
	
	str := concat(str, ANY_TO_STRING(gvl.gMagicNum));	
	str := concat(str, ANY_TO_STRING(","));
	check_sum := check_sum + gvl.gMagicNum;
	
	str := concat(str, ANY_TO_STRING(check_sum));		
	str := concat(str, ANY_TO_STRING(";"));
	
	str := concat(str, ANY_TO_STRING("$R$N"));		
	str_size := ANY_TO_DWORD(len(str));
	
	udiByteWrite := sysfile.SysFileWrite(hFile := hFile,pbyBuffer := ADR(str),ulSize := str_size, pResult := ADR(udiWriteError));
	sysfile.SysFileClose(hFile);
	fn_write_para_file := TRUE;
END_IF

END_FUNCTION

// Changsha_Xiangji_ARM_Cortex_A9_xilinx_zynq7000_linux/Application/parameters/fn_read_para_file
FUNCTION fn_read_para_file : BOOL
VAR_INPUT
	pPara :POINTER TO ST_PARA;
END_VAR
VAR
	hFile: RTS_IEC_HANDLE;
	udiOpenError: RTS_IEC_RESULT;
	udiReadError: RTS_IEC_RESULT;
	i :INT;
	iTemp: UDINT;
	udiPos: UDINT;
	str: STRING(65535);
	str_size: __XWORD;
	udiByteRead: __XWORD;

	len_of_line: INT;
	len_of_number :INT;
	magicNumber:REAL;
	check_sum:REAL:= 0;
	temp_num:REAL;
END_VAR

fn_read_para_file := FALSE;

//检测文件是否存在
hFile := sysfileopen(szFile := gvl.para_file, am := sysfile.AM_READ, pResult:= ADR(udiOpenError));
IF hFile = RTS_INVALID_HANDLE	THEN  //文件不存在
	RETURN;
END_IF

//文件存在，开始读取内容
udiPos := SysFileSetPos(hFile:=hFile, ulOffset := 0);
udiByteRead := sysfile.SysFileRead(hfile := hFile,pbyBuffer := ADR(str), ulSize := SIZEOF(str), pResult := ADR(udiReadError));
IF udiByteRead < 4 THEN  //读取失败
	sysfile.SysFileClose(hFile := hFile);
	RETURN;
END_IF
//根据“;“的位置确定本行的长度
len_of_line := find(str,WSTRING_TO_STRING(";"));
iTemp := iTemp + INT_TO_UDINT(len_of_line) + 2;  //加上换行和回车符的长度

//读取本行的数字
check_sum := 0;
FOR i := 0 TO pPara^.len DO
	len_of_number := find(str, WSTRING_TO_STRING(","));
	temp_num := STRING_TO_REAL(left(str,len_of_number-1));
	check_sum := check_sum + temp_num;
	pPara^.para_val[i] := temp_num;
	str := delete(str, len_of_number,1);	
END_FOR

len_of_number := find(str, WSTRING_TO_STRING(","));
temp_num := STRING_TO_REAL(left(str,len_of_number-1));
check_sum := check_sum + temp_num;		
magicNumber := temp_num;		
str := delete(str, len_of_number,1);

len_of_number := find(str, WSTRING_TO_STRING(";"));   //最后一个校验和后面是“;”
temp_num := STRING_TO_REAL(left(str,len_of_number-1));
str := delete(str, len_of_number,1);
sysfile.SysFileClose(hFile := hFile);
IF ABS(check_sum - temp_num) > 0.01 THEN  //校验错
	RETURN;
END_IF

IF ABS(magicNumber - gvl.gMagicNum) > 0.01 THEN  //两个浮点数不相等
	RETURN;		
END_IF

pPara^.para_ok := TRUE;

fn_read_para_file := TRUE;
RETURN;

END_FUNCTION

// Changsha_Xiangji_ARM_Cortex_A9_xilinx_zynq7000_linux/Application/Falsh_RW
PROGRAM Falsh_RW
VAR
	bFlashW: BOOL := true;
	bFlashR1: BOOL := true;
	iStat:UINT:= 0;
END_VAR

CASE iStat OF
	0: //init
	fn_read_para_file(ADR(g_parameters));
	(*IF NOT g_parameters.para_ok THEN  //读取参数失败，设置初始值
			g_parameters.para_val[0] := 50;//加减值
			g_parameters.para_val[1] := 850;//最低转速
			g_parameters.para_val[2] := 1450;//标准转速
			g_parameters.para_val[3] := 1750;//强力转速
			g_parameters.para_val[4] := 0;//扫盘转速
			g_parameters.para_val[5] := 1850;//高压水泵超速报警
			g_parameters.para_val[6] := 1950;//高压水泵超速停止
			g_parameters.para_val[7] := 2500;//最高转速
			g_parameters.para_val[8] := 850;//怠速
			g_parameters.para_val[9] := 1000;//清洁低速
			g_parameters.para_val[10] := 1000;//清洁中低速
			g_parameters.para_val[11] := 1100;//清洁中高速
			g_parameters.para_val[12] := 1450;//清洁高速
			g_parameters.para_val[13] := 1200;//一般低速
			g_parameters.para_val[14] := 1350;//一般中低速
			g_parameters.para_val[15] := 1500;//一般中高速
			g_parameters.para_val[16] := 1750;//一般高速
			g_parameters.para_val[17] := 1350;//污染低速
			g_parameters.para_val[18] := 1550;//污染中低速
			g_parameters.para_val[19] := 1750;//污染中高速
			g_parameters.para_val[20] := 1750;//污染高速
			g_parameters.para_val[21] := 100;
			g_parameters.para_ok := TRUE;
			fn_write_para_file(g_parameters);
			ELSE *)
	        S_IncDec_Speed:=ANY_TO_UINT(g_parameters.para_val[0]) ;//加减值
            S_min_speed:=ANY_TO_UINT(g_parameters.para_val[1]) ;//最低转速
	        S_Standard_Speed:=ANY_TO_UINT(g_parameters.para_val[2]);//标准转速
	        S_Strong_Speed:=ANY_TO_UINT(g_parameters.para_val[3]) ;//强力转速
	        S_Sweep_Speed:=ANY_TO_UINT(g_parameters.para_val[4]);//扫盘转速
	        S_Pumpspeed_arm:=ANY_TO_UINT(g_parameters.para_val[5]);//高压水泵超速报警
	        S_Pumpspeed_stop:=ANY_TO_UINT(g_parameters.para_val[6]);//高压水泵超速停止
	        S_MAX_Speed:=ANY_TO_UINT(g_parameters.para_val[7]);//最高转速
	        S_Idle_Speed:=ANY_TO_UINT(g_parameters.para_val[8]);//怠速
	        S_clean_low_speed:=ANY_TO_UINT(g_parameters.para_val[9]);//清洁低速
	        S_clean_midlow_speed:=ANY_TO_UINT(g_parameters.para_val[10]);//清洁中低速
	        S_clean_midhigh_speed:=ANY_TO_UINT(g_parameters.para_val[11]);//清洁中高速
	        S_clean_high_speed:=ANY_TO_UINT(g_parameters.para_val[12]);//清洁高速
	        S_normal_low_speed:=ANY_TO_UINT(g_parameters.para_val[13]);//一般低速
	        S_normal_midlow_speed:=ANY_TO_UINT(g_parameters.para_val[14]);//一般中低速
	        S_normal_midhigh_speed:=ANY_TO_UINT(g_parameters.para_val[15]);//一般中高速
	        S_normal_high_speed:=ANY_TO_UINT(g_parameters.para_val[16]);//一般高速
	        S_dirty_low_speed:=ANY_TO_UINT(g_parameters.para_val[17]);//污染低速
	        S_dirty_midlow_speed:=ANY_TO_UINT(g_parameters.para_val[18]);//污染中低速
	        S_dirty_midhigh_speed:=ANY_TO_UINT(g_parameters.para_val[19]);//污染中高速
	        S_dirty_high_speed:=ANY_TO_UINT(g_parameters.para_val[20]);//污染高速	
			motor_work_time:=ANY_TO_DWORD(g_parameters.para_val[22])+ANY_TO_DWORD(g_parameters.para_val[23])*16#100+ANY_TO_DWORD(g_parameters.para_val[24])*16#10000+ANY_TO_DWORD(g_parameters.para_val[25])*16#1000000;	
    
		iSTat := 10;

	10:
	
END_CASE
(*//读取参数失败，设置初始值
IF NOT g_parameters.para_ok THEN  //读取参数失败，设置初始值
			g_parameters.para_val[0] := 50;//加减值
			g_parameters.para_val[1] := 850;//最低转速
			g_parameters.para_val[2] := 1450;//标准转速
			g_parameters.para_val[3] := 1750;//强力转速
			g_parameters.para_val[4] := 0;//扫盘转速
			g_parameters.para_val[5] := 1850;//高压水泵超速报警
			g_parameters.para_val[6] := 1950;//高压水泵超速停止
			g_parameters.para_val[7] := 2500;//最高转速
			g_parameters.para_val[8] := 850;//怠速
			g_parameters.para_val[9] := 1000;//清洁低速
			g_parameters.para_val[10] := 1000;//清洁中低速
			g_parameters.para_val[11] := 1100;//清洁中高速
			g_parameters.para_val[12] := 1450;//清洁高速
			g_parameters.para_val[13] := 1200;//一般低速
			g_parameters.para_val[14] := 1350;//一般中低速
			g_parameters.para_val[15] := 1500;//一般中高速
			g_parameters.para_val[16] := 1750;//一般高速
			g_parameters.para_val[17] := 1350;//污染低速
			g_parameters.para_val[18] := 1550;//污染中低速
			g_parameters.para_val[19] := 1750;//污染中高速
			g_parameters.para_val[20] := 1750;//污染高速
			g_parameters.para_val[21] := 100;
			g_parameters.para_ok := TRUE;
			fn_write_para_file(g_parameters);
END_IF	
*)



//********HMI写参数
IF Re_IncDec_Speed>0 AND S_IncDec_Speed<>Re_IncDec_Speed THEN
	g_parameters.para_val[0] := Re_IncDec_Speed;//加减值
	fn_write_para_file(g_parameters);
    S_IncDec_Speed :=ANY_TO_UINT(g_parameters.para_val[0]);   
END_IF
//********HMI写参数
IF Re_motor_min_speed>0 AND S_min_speed<>Re_motor_min_speed THEN
	g_parameters.para_val[1] := Re_motor_min_speed;//最低转速
	fn_write_para_file(g_parameters);
    S_min_speed :=ANY_TO_UINT(g_parameters.para_val[1]);   
END_IF
//********HMI写参数
IF Re_normal_speed>0 AND S_Standard_Speed<>Re_normal_speed THEN
	g_parameters.para_val[2] := Re_normal_speed;//标准转速
	fn_write_para_file(g_parameters);
    S_Standard_Speed :=ANY_TO_UINT(g_parameters.para_val[2]);   
END_IF
//********HMI写参数
IF Re_strong_Speed>0 AND S_Strong_Speed<>Re_strong_Speed THEN
	g_parameters.para_val[3] := Re_strong_Speed;//强力转速
	fn_write_para_file(g_parameters);
    S_Strong_Speed :=ANY_TO_UINT(g_parameters.para_val[3]);   
END_IF
//********HMI写参数
IF S_Idle_Speed>0 AND ((Re_Sweep_Speed=0) OR (Re_Sweep_Speed=1) OR (Re_Sweep_Speed=2)) AND Re_Sweep_Speed<>S_Sweep_Speed THEN
	g_parameters.para_val[4] := Re_Sweep_Speed;//扫盘转速
	fn_write_para_file(g_parameters);
    S_Sweep_Speed :=ANY_TO_UINT(g_parameters.para_val[4]);   
END_IF
//********HMI写参数
IF Re_Pumpspeed_arm>0 AND S_Pumpspeed_arm<>Re_Pumpspeed_arm THEN
	g_parameters.para_val[5] := Re_Pumpspeed_arm;//高压水泵超速报警
	fn_write_para_file(g_parameters);
    S_Pumpspeed_arm :=ANY_TO_UINT(g_parameters.para_val[5]);   
END_IF
//********HMI写参数
IF Re_Pumpspeed_stop>0 AND S_Pumpspeed_stop<>Re_Pumpspeed_stop THEN
	g_parameters.para_val[6] := Re_Pumpspeed_stop;//高压水泵超速停止
	fn_write_para_file(g_parameters);
    S_Pumpspeed_stop :=ANY_TO_UINT(g_parameters.para_val[6]);   
END_IF
//********HMI写参数
IF Re_MAX_Speed>0 AND S_MAX_Speed<>Re_MAX_Speed THEN
	g_parameters.para_val[7] := Re_MAX_Speed;//最高转速
	fn_write_para_file(g_parameters);
    S_MAX_Speed :=ANY_TO_UINT(g_parameters.para_val[7]);   
END_IF
//********HMI写参数
IF Re_Idle_Speed>0 AND S_Idle_Speed<>Re_Idle_Speed THEN
	g_parameters.para_val[8] := Re_Idle_Speed;//怠速
	fn_write_para_file(g_parameters);
    S_Idle_Speed :=ANY_TO_UINT(g_parameters.para_val[8]);   
END_IF
//********HMI写参数
IF Re_clean_low_speed>0 AND S_clean_low_speed<>Re_clean_low_speed THEN
	g_parameters.para_val[9] := Re_clean_low_speed;//清洁低速
	fn_write_para_file(g_parameters);
    S_clean_low_speed :=ANY_TO_UINT(g_parameters.para_val[9]);   
END_IF
//********HMI写参数
IF Re_clean_midlow_speed>0 AND S_clean_midlow_speed<>Re_clean_midlow_speed THEN
	g_parameters.para_val[10] := Re_clean_midlow_speed;//清洁中低速
	fn_write_para_file(g_parameters);
    S_clean_midlow_speed :=ANY_TO_UINT(g_parameters.para_val[10]);   
END_IF
//********HMI写参数
IF Re_clean_midhigh_speed>0 AND S_clean_midhigh_speed<>Re_clean_midhigh_speed THEN
	g_parameters.para_val[11] := Re_clean_midhigh_speed;//清洁中高速
	fn_write_para_file(g_parameters);
    S_clean_midhigh_speed :=ANY_TO_UINT(g_parameters.para_val[11]);   
END_IF
//********HMI写参数
IF Re_clean_high_speed>0 AND S_clean_high_speed<>Re_clean_high_speed THEN
	g_parameters.para_val[12] := Re_clean_high_speed;//清洁高速
	fn_write_para_file(g_parameters);
    S_clean_high_speed :=ANY_TO_UINT(g_parameters.para_val[12]);   
END_IF
//********HMI写参数
IF Re_normal_low_speed>0 AND S_normal_low_speed<>Re_normal_low_speed THEN
	g_parameters.para_val[13] := Re_normal_low_speed;//一般低速
	fn_write_para_file(g_parameters);
    S_normal_low_speed :=ANY_TO_UINT(g_parameters.para_val[13]);   
END_IF
//********HMI写参数
IF Re_normal_midlow_speed>0 AND S_normal_midlow_speed<>Re_normal_midlow_speed THEN
	g_parameters.para_val[14] := Re_normal_midlow_speed;//一般中低速
	fn_write_para_file(g_parameters);
    S_normal_midlow_speed :=ANY_TO_UINT(g_parameters.para_val[14]);   
END_IF
//********HMI写参数
IF Re_normal_midhigh_speed>0 AND S_normal_midhigh_speed<>Re_normal_midhigh_speed THEN
	g_parameters.para_val[15] := Re_normal_midhigh_speed;//一般中高速
	fn_write_para_file(g_parameters);
    S_normal_midhigh_speed :=ANY_TO_UINT(g_parameters.para_val[15]);   
END_IF
//********HMI写参数
IF Re_normal_high_speed>0 AND S_normal_high_speed<>Re_normal_high_speed THEN
	g_parameters.para_val[16] := Re_normal_high_speed;//一般高速
	fn_write_para_file(g_parameters);
    S_normal_high_speed :=ANY_TO_UINT(g_parameters.para_val[16]);   
END_IF
//********HMI写参数
IF Re_dirty_low_speed>0 AND S_dirty_low_speed<>Re_dirty_low_speed THEN
	g_parameters.para_val[17] := Re_dirty_low_speed;//污染低速
	fn_write_para_file(g_parameters);
    S_dirty_low_speed :=ANY_TO_UINT(g_parameters.para_val[17]);   
END_IF
//********HMI写参数
IF Re_dirty_midlow_speed>0 AND S_dirty_midlow_speed<>Re_dirty_midlow_speed THEN
	g_parameters.para_val[18] := Re_dirty_midlow_speed;//污染中低速
	fn_write_para_file(g_parameters);
    S_dirty_midlow_speed :=ANY_TO_UINT(g_parameters.para_val[18]);   
END_IF
//********HMI写参数
IF Re_dirty_midhigh_speed>0 AND S_dirty_midhigh_speed<>Re_dirty_midhigh_speed THEN
	g_parameters.para_val[19] := Re_dirty_midhigh_speed;//污染中高速
	fn_write_para_file(g_parameters);
    S_dirty_midhigh_speed :=ANY_TO_UINT(g_parameters.para_val[19]);   
END_IF
//********HMI写参数
IF Re_dirty_high_speed>0 AND S_dirty_high_speed<>Re_dirty_high_speed THEN
	g_parameters.para_val[20] := Re_dirty_high_speed;//污染高速
	fn_write_para_file(g_parameters);
    S_dirty_high_speed :=ANY_TO_UINT(g_parameters.para_val[20]);   
END_IF





(*首次上电写一次参数组，后面再也不写参数组*)
IF bFlashW AND NOT (g_parameters.para_val[21]=100) THEN
    bFlashW:=FALSE;
    g_parameters.para_val[0] := 50;//加减值
    g_parameters.para_val[1] := 850;//最低转速
	g_parameters.para_val[2] := 1450;//标准转速
	g_parameters.para_val[3] := 1750;//强力转速
	g_parameters.para_val[4] := 0;//扫盘转速
	g_parameters.para_val[5] := 1850;//高压水泵超速报警
	g_parameters.para_val[6] := 1950;//高压水泵超速停止
	g_parameters.para_val[7] := 2500;//最高转速
	g_parameters.para_val[8] := 850;//怠速
	g_parameters.para_val[9] := 1000;//清洁低速
	g_parameters.para_val[10] := 1000;//清洁中低速
	g_parameters.para_val[11] := 1100;//清洁中高速
	g_parameters.para_val[12] := 1450;//清洁高速
	g_parameters.para_val[13] := 1200;//一般低速
	g_parameters.para_val[14] := 1350;//一般中低速
	g_parameters.para_val[15] := 1500;//一般中高速
	g_parameters.para_val[16] := 1750;//一般高速
	g_parameters.para_val[17] := 1350;//污染低速
	g_parameters.para_val[18] := 1550;//污染中低速
	g_parameters.para_val[19] := 1750;//污染中高速
	g_parameters.para_val[20] := 1750;//污染高速
	g_parameters.para_val[21] := 0;
	g_parameters.para_val[22] := 0;
	g_parameters.para_val[23] := 0;
	g_parameters.para_val[24] := 0;
	g_parameters.para_val[25] := 0;
	g_parameters.para_ok := TRUE;
	fn_write_para_file(g_parameters);
	
	fn_read_para_file(ADR(g_parameters));
	S_IncDec_Speed:=ANY_TO_UINT(g_parameters.para_val[0]) ;//加减值
    S_min_speed:=ANY_TO_UINT(g_parameters.para_val[1]) ;//最低转速
	S_Standard_Speed:=ANY_TO_UINT(g_parameters.para_val[2]);//标准转速
	S_Strong_Speed:=ANY_TO_UINT(g_parameters.para_val[3]) ;//强力转速
	S_Sweep_Speed:=ANY_TO_UINT(g_parameters.para_val[4]);//扫盘转速
	S_Pumpspeed_arm:=ANY_TO_UINT(g_parameters.para_val[5]);//高压水泵超速报警
	S_Pumpspeed_stop:=ANY_TO_UINT(g_parameters.para_val[6]);//高压水泵超速停止
	S_MAX_Speed:=ANY_TO_UINT(g_parameters.para_val[7]);//最高转速
	S_Idle_Speed:=ANY_TO_UINT(g_parameters.para_val[8]);//怠速
	S_clean_low_speed:=ANY_TO_UINT(g_parameters.para_val[9]);//清洁低速
	S_clean_midlow_speed:=ANY_TO_UINT(g_parameters.para_val[10]);//清洁中低速
	S_clean_midhigh_speed:=ANY_TO_UINT(g_parameters.para_val[11]);//清洁中高速
	S_clean_high_speed:=ANY_TO_UINT(g_parameters.para_val[12]);//清洁高速
	S_normal_low_speed:=ANY_TO_UINT(g_parameters.para_val[13]);//一般低速
	S_normal_midlow_speed:=ANY_TO_UINT(g_parameters.para_val[14]);//一般中低速
	S_normal_midhigh_speed:=ANY_TO_UINT(g_parameters.para_val[15]);//一般中高速
	S_normal_high_speed:=ANY_TO_UINT(g_parameters.para_val[16]);//一般高速
	S_dirty_low_speed:=ANY_TO_UINT(g_parameters.para_val[17]);//污染低速
	S_dirty_midlow_speed:=ANY_TO_UINT(g_parameters.para_val[18]);//污染中低速
	S_dirty_midhigh_speed:=ANY_TO_UINT(g_parameters.para_val[19]);//污染中高速
	S_dirty_high_speed:=ANY_TO_UINT(g_parameters.para_val[20]);//污染高速
 
END_IF

END_PROGRAM

// Changsha_Xiangji_ARM_Cortex_A9_xilinx_zynq7000_linux/Application/DO_fault
PROGRAM DO_fault
VAR

	do_fault_02 :FB_DOH_FAULT;  //创建故障诊断功能块的实例，每个DO端口创建一个
	do_fault_03 :FB_DOH_FAULT;  //创建故障诊断功能块的实例，每个DO端口创建一个	
	do_fault_04 :FB_DOH_FAULT;  //创建故障诊断功能块的实例，每个DO端口创建一个
	do_fault_05 :FB_DOH_FAULT;  //创建故障诊断功能块的实例，每个DO端口创建一个
	do_fault_06 :FB_DOH_FAULT;  //创建故障诊断功能块的实例，每个DO端口创建一个
	do_fault_07 :FB_DOH_FAULT;  //创建故障诊断功能块的实例，每个DO端口创建一个
	do_fault_08 :FB_DOH_FAULT;  //创建故障诊断功能块的实例，每个DO端口创建一个
	do_fault_09 :FB_DOH_FAULT;  //创建故障诊断功能块的实例，每个DO端口创建一个
	do_fault_10 :FB_DOH_FAULT;  //创建故障诊断功能块的实例，每个DO端口创建一个
	do_fault_11 :FB_DOH_FAULT;  //创建故障诊断功能块的实例，每个DO端口创建一个
	do_fault_12 :FB_DOH_FAULT;  //创建故障诊断功能块的实例，每个DO端口创建一个
	do_fault_13 :FB_DOH_FAULT;  //创建故障诊断功能块的实例，每个DO端口创建一个
	do_fault_16 :FB_DOH_FAULT;  //创建故障诊断功能块的实例，每个DO端口创建一个
    do_fault_17 :FB_DOH_FAULT;  //创建故障诊断功能块的实例，每个DO端口创建一个
    do_fault_18 :FB_DOH_FAULT;  //创建故障诊断功能块的实例，每个DO端口创建一个	
    do_fault_19 :FB_DOH_FAULT;  //创建故障诊断功能块的实例，每个DO端口创建一个
    do_fault_20 :FB_DOH_FAULT;  //创建故障诊断功能块的实例，每个DO端口创建一个
    do_fault_21 :FB_DOH_FAULT;  //创建故障诊断功能块的实例，每个DO端口创建一个
    do_fault_22 :FB_DOH_FAULT;  //创建故障诊断功能块的实例，每个DO端口创建一个
    do_fault_23 :FB_DOH_FAULT;  //创建故障诊断功能块的实例，每个DO端口创建一个
	do_fault_28 :FB_DOH_FAULT;  //创建故障诊断功能块的实例，每个DO端口创建一个
	do_fault_29 :FB_DOH_FAULT;  //创建故障诊断功能块的实例，每个DO端口创建一个
	do_fault_30 :FB_DOH_FAULT;  //创建故障诊断功能块的实例，每个DO端口创建一个
	do_fault_31 :FB_DOH_FAULT;  //创建故障诊断功能块的实例，每个DO端口创建一个


END_VAR

//左扫盘降
do_fault_03(enable := TRUE,dout := DO_Lsweep_down, ai := ai_21);
DO_Lsweep_down_short := do_fault_03.short;
DO_Lsweep_down_open := do_fault_03.open;
//左扫盘升
do_fault_04(enable := TRUE,dout := DO_Lsweep_up, ai := ai_22);
DO_Lsweep_up_short := do_fault_04.short;
DO_Lsweep_up_open := do_fault_04.open;
//右扫盘降
do_fault_05(enable := TRUE,dout := DO_Rsweep_down, ai := ai_23);
DO_Rsweep_down_short := do_fault_05.short;
DO_Rsweep_down_open := do_fault_05.open;
//右扫盘升
do_fault_06(enable := TRUE,dout := DO_Rsweep_up, ai := ai_24);
DO_Rsweep_up_short := do_fault_06.short;
DO_Rsweep_up_open := do_fault_06.open;
//左扫摆出
do_fault_07(enable := TRUE,dout := DO_Lsweep_out, ai := ai_25);
DO_Lsweep_out_short := do_fault_07.short;
DO_Lsweep_out_open := do_fault_07.open;
//右扫摆出
do_fault_08(enable := TRUE,dout := DO_Rsweep_out, ai := ai_26);
DO_Rsweep_out_short := do_fault_08.short;
DO_Rsweep_out_open := do_fault_08.open;
//左喷杆摆出
do_fault_09(enable := TRUE,dout := DO_Lrod_out, ai := ai_27);
DO_Lrod_out_short := do_fault_09.short;
DO_Lrod_out_open := do_fault_09.open;
//右喷杆摆出
do_fault_10(enable := TRUE,dout := DO_Rrod_out, ai := ai_28);
DO_Rrod_out_short := do_fault_10.short;
DO_Rrod_out_open := do_fault_10.open;
(*//点喷上
do_fault_11(enable := TRUE,dout := DO_pointshoot_up, ai := ai_29);
DO_pointshoot_up_short := do_fault_11.short;
DO_pointshoot_up_open := do_fault_11.open;
//点喷下
do_fault_02(enable := TRUE,dout := DO_pointshoot_Down, ai := ai_20);
DO_pointshoot_Down_short := do_fault_02.short;
DO_pointshoot_Down_open := do_fault_02.open;
//点喷左
do_fault_28(enable := TRUE,dout := DO_pointshoot_left, ai := ai_21);
DO_pointshoot_left_short := do_fault_28.short;
DO_pointshoot_left_open := do_fault_28.open;
//点喷右
do_fault_28(enable := TRUE,dout := DO_pointshoot_right, ai := ai_21);
DO_pointshoot_right_short := do_fault_28.short;
DO_pointshoot_right_open := do_fault_28.open;*)
//备用
//do_fault_25(enable := TRUE,dout := DO_pointshoot_right, ai := ai_21);
//DO_pointshoot_right_short := do_fault_25.short;
//DO_pointshoot_right_open := do_fault_25.open;
//水泵卸荷球阀
do_fault_23(enable := TRUE,dout := DO_water_overflow, ai := ai_41);
DO_water_overflow_short := do_fault_28.short;
DO_water_overflow_open := do_fault_28.open;
//左侧喷杆球阀
do_fault_22(enable := TRUE,dout := DO_Lrod_water, ai := ai_40);
DO_Lrod_water_short := do_fault_22.short;
DO_Lrod_water_open := do_fault_22.open;
//右侧喷杆球阀
do_fault_21(enable := TRUE,dout := DO_Rrod_water, ai := ai_39);
DO_Rrod_water_short := do_fault_21.short;
DO_Rrod_water_open := do_fault_21.open;
//吸嘴喷杆球阀
do_fault_20(enable := TRUE,dout := DO_Suction_water, ai := ai_38);
DO_Suction_water_short := do_fault_20.short;
DO_Suction_water_open := do_fault_20.open;
//喷雾球阀
do_fault_19(enable := TRUE,dout := DO_Hpressure_water, ai := ai_37);
DO_Hpressure_water_short := do_fault_19.short;
DO_Hpressure_water_open := do_fault_19.open;
//自洁喷杆球阀
do_fault_18(enable := TRUE,dout := DO_selfclean_water, ai := ai_36);
DO_selfclean_water_short := do_fault_18.short;
DO_selfclean_water_open := do_fault_18.open;
//水泵离合器啮合
do_fault_17(enable := TRUE,dout := DO_Hpre_pump, ai := ai_35);
DO_Hpre_pump_short := do_fault_17.short;
DO_Hpre_pump_open := do_fault_17.open;
//低压隔膜泵
do_fault_16(enable := TRUE,dout := DO_fog_Spump, ai := ai_34);
DO_fog_Spump_short := do_fault_16.short;
DO_fog_Spump_open := do_fault_16.open;
//电机使能
//do_fault_13(enable := TRUE,dout := DO_Motor_en, ai := ai_31);
//DO_Motor_en_short := do_fault_13.short;
//DO_Motor_en_open := do_fault_13.open;
(*//水冷泵电机
do_fault_30(enable := TRUE,dout := DO_watercooler_pump, ai := ai_21);
DO_watercooler_pump_short := do_fault_30.short;
DO_watercooler_pump_open := do_fault_30.open;
//散热风扇
do_fault_31(enable := TRUE,dout := DO_cooler_fan, ai := ai_21);
DO_cooler_fan_short := do_fault_31.short;
DO_cooler_fan_open := do_fault_31.open;*)
(*//备用动力控制
do_fault_12(enable := TRUE,dout := DO_backup_power, ai := ai_30);
DO_backup_power_short := do_fault_12.short;
DO_backup_power_open := do_fault_12.open;
*)

END_PROGRAM

// Changsha_Xiangji_ARM_Cortex_A9_xilinx_zynq7000_linux/Application/funcs/FB_DOH_FAULT
FUNCTION_BLOCK FB_DOH_FAULT      //检测MIC7000系列控制器高有效输出端口的短路和短线故障 功能块
VAR_INPUT
	enable :BOOL;   //开关，true 表示启用本功能块
	dout:BOOL;     	//需要检测的高有效开关量输出端口值
	ai:DWORD;      	//需要检测的高有效输出端口对应的模拟量输入值
END_VAR
VAR_OUTPUT
	ok:BOOL;    	//正常标志，为true表示无故障
	short:BOOL;  	//短路故障标志
	open:BOOL;    	//短线故障标志
END_VAR

VAR
	stat: DWORD := 0;
	stat_short :DWORD := 0;
	stat_open :DWORD := 0;
	short_cntr :DWORD := 0;
	open_cntr :DWORD := 0;
END_VAR

VAR CONSTANT   //参数定义，可以根据情况修改
	SHORT_VALUE :DWORD := 3000; //短路门槛值
	OPEN_VALUE :DWORD := 25;   	//开路门槛值
	TIME_OUT :DWORD := 10;   	//超时周期数
END_VAR

IF NOT enable THEN
	ok := TRUE;
	short := FALSE;
	open := FALSE;
	RETURN;
END_IF

CASE stat OF
	0:
		ok := TRUE;
		short := FALSE;
		open := FALSE;
		IF dout THEN  
			stat := 100;	// dout high, detect short
			stat_short := 0;
		ELSE 
			stat := 200;  //dout low, detect open
			stat_open := 0;
		END_IF
	
	100:  //detect short
		IF NOT dout THEN  //return 
			stat := 0;
		END_IF
		CASE stat_short OF
			0:
				short := FALSE;
				IF ai < SHORT_VALUE THEN  //short
					stat_short := 10;
					short_cntr := 0;
				END_IF
			10:  //short wait for timeout
				IF ai > SHORT_VALUE THEN  //normal , wait for return
					IF short_cntr = 0 THEN
						stat_short := 0;
					ELSE
						short_cntr := short_cntr - 1;
					END_IF
				ELSE  //short, 
					IF short_cntr > TIME_OUT THEN
						short := TRUE;
					ELSE
						short_cntr := short_cntr + 1;
					END_IF		
				END_IF	
		END_CASE

	200:
		IF dout THEN  //  dout high, return to detect short
			stat := 0;
		END_IF
		CASE stat_open OF
			0:
				open := FALSE;
				IF ai > OPEN_VALUE THEN  //open
					stat_open := 10;
					open_cntr := 0;
				END_IF
			10:
				IF ai < OPEN_VALUE THEN  //normal, wait for return
					IF open_cntr = 0 THEN
						stat_open := 0;
					ELSE
						open_cntr := open_cntr - 1;
					END_IF
				ELSE
					IF open_cntr > TIME_OUT THEN
						open := TRUE;
					ELSE
						open_cntr := open_cntr + 1;
					END_IF
				END_IF			
		END_CASE
END_CASE

ok := (NOT short) AND (NOT open);

END_FUNCTION_BLOCK

// Changsha_Xiangji_ARM_Cortex_A9_xilinx_zynq7000_linux/Application/Test
PROGRAM Test
VAR
	
	// 水冷泵测试上升沿
	R_Test_watercooler_pump: R_TRIG;
	cooler_motor_Test1: BOOL;
	// 散热风扇上升沿
	R_Test_cooler_fan: R_TRIG;
	cooler_fan_Test1: BOOL;
	// 扫盘中速上升沿
	R_Test_Sweep_Mspeed: R_TRIG;
	Sweep_Mspeed_Test1: BOOL;
	// 扫盘低速上升沿
	R_Test_Sweep_Lspeed: R_TRIG;
	Sweep_Lspeed_Test1: BOOL;
	// 左扫旋转测试上升沿
	R_Test_LSweep: R_TRIG;
	LSweep_Test1: BOOL;
	// 右扫旋转测试上升沿
	R_Test_RSweep: R_TRIG;
	RSweep_Test1: BOOL;
	// 全扫旋转测试上升沿
	R_Test_ASweep: R_TRIG;
	ASweep_Test1: BOOL;
	// 左扫摆出测试上升沿
	R_Test_LSweep_out: R_TRIG;
	LSweep_out_Test1: BOOL;
	// 右扫盘摆出测试上升沿
	R_Test_RSweep_out: R_TRIG;
	RSweep_out_Test1: BOOL;
	// 左喷杆摆出测试上升沿
	R_Test_Lrod_OUT: R_TRIG;
	Lrod_OUT_Test1: BOOL;
	// 右喷杆摆出测试上升沿
	R_Test_Rrod_OUT: R_TRIG;
	Rrod_OUT_Test1: BOOL;
	// 左喷杆喷水测试上升沿
	R_Test_Lrod_water: R_TRIG;
	Lrod_water_Test1: BOOL;
	// 右喷杆喷水测试上升沿
	R_Test_Rrod_water: R_TRIG;
	Rrod_water_Test1: BOOL;
	// 吸嘴喷杆喷水测试上升沿
	R_Test_Suction_water: R_TRIG;
	Suction_water_Test1: BOOL;
	// 高压冲洗测试上升沿
	R_Test_Hpre_wash: R_TRIG;
	Hpre_wash_Test1: BOOL;
	// 自洁测试上升沿
	R_Test_selfclean: R_TRIG;
	selfclean_water_Test1: BOOL;
	// 高压水泵啮合测试上升沿
	R_Test_Hpre_pump_gearin: R_TRIG;
	Hpress_pump_gearin_Test1: BOOL;
	T_pumpClutch: Ton;
	// 喷雾降尘泵测试上升沿
	R_Test_fogpump: R_TRIG;
	Fog_pump_Test1: BOOL;
	T_Fog_pump_Test: Ton;
	// 污水泵测试上升沿
	R_Test_wastewater_pump: R_TRIG;
	Wastewater_pump_Test1: BOOL;
	// 污水泵球阀测试上升沿
	R_Test_wastewater_valve: R_TRIG;
	Wastewater_valve_Test1: BOOL;
	// 备用动力测试上升沿
	R_Test_backup_power: R_TRIG;
	Backup_power_Test1: BOOL;
	T_Backup_power_Test: Ton;
	

END_VAR

